  PROC DrawPart24()
    MoveL Offs(pOrigin,272.74,80.44,0.00),v40,z0,tPen\WObj:=wPaper;
    MoveL Offs(pOrigin,271.25,97.44,0.00),v40,z0,tPen\WObj:=wPaper;
    MoveL Offs(pOrigin,271.04,102.96,0.00),v40,z0,tPen\WObj:=wPaper;
    MoveL Offs(pOrigin,271.25,114.65,0.00),v40,z0,tPen\WObj:=wPaper;
    MoveL Offs(pOrigin,272.95,133.56,0.00),v40,z0,tPen\WObj:=wPaper;
    MoveL Offs(pOrigin,275.92,151.84,0.00),v40,z0,tPen\WObj:=wPaper;
    MoveL Offs(pOrigin,275.71,152.69,0.00),v40,z0,tPen\WObj:=wPaper;
    MoveL Offs(pOrigin,275.71,152.69,0.00),v40,z0,tPen\WObj:=wPaper;
    MoveL Offs(pOrigin,276.35,154.39,0.00),v40,z0,tPen\WObj:=wPaper;
    MoveL Offs(pOrigin,280.39,173.73,0.00),v40,z0,tPen\WObj:=wPaper;
    MoveL Offs(pOrigin,280.39,175.43,0.00),v40,z0,tPen\WObj:=wPaper;
    MoveL Offs(pOrigin,281.24,177.12,0.00),v40,z0,tPen\WObj:=wPaper;
    MoveL Offs(pOrigin,286.76,199.01,0.00),v40,z0,tPen\WObj:=wPaper;
    MoveL Offs(pOrigin,286.76,199.01,0.00),v40,z0,tPen\WObj:=wPaper;
    MoveL Offs(pOrigin,288.25,206.66,0.00),v40,z0,tPen\WObj:=wPaper;
    MoveL Offs(pOrigin,289.10,213.46,0.00),v40,z0,tPen\WObj:=wPaper;
    MoveL Offs(pOrigin,289.10,221.32,0.00),v40,z0,tPen\WObj:=wPaper;
    MoveL Offs(pOrigin,288.82,222.39,0.00),v40,z0,tPen\WObj:=wPaper;
    MoveL Offs(pOrigin,288.25,222.81,0.00),v40,fine,tPen\WObj:=wPaper;
    MoveL Offs(pOrigin,288.25,222.81,6.00),v60,z5,tPen\WObj:=wPaper;
    MoveL Offs(pOrigin,287.19,224.30,6.00),vTravel,z5,tPen\WObj:=wPaper;
    MoveL Offs(pOrigin,287.19,224.30,0.00),v60,z0,tPen\WObj:=wPaper;
    MoveL Offs(pOrigin,287.61,224.51,0.00),v40,z0,tPen\WObj:=wPaper;
    MoveL Offs(pOrigin,287.19,224.30,0.00),v40,fine,tPen\WObj:=wPaper;
    MoveL Offs(pOrigin,287.19,224.30,6.00),v60,z5,tPen\WObj:=wPaper;
    MoveL Offs(pOrigin,296.11,217.29,6.00),vTravel,z5,tPen\WObj:=wPaper;
    MoveL Offs(pOrigin,296.11,217.29,0.00),v60,z0,tPen\WObj:=wPaper;
    MoveL Offs(pOrigin,294.41,218.99,0.00),v40,z0,tPen\WObj:=wPaper;
    MoveL Offs(pOrigin,296.11,217.29,0.00),v40,fine,tPen\WObj:=wPaper;
    MoveL Offs(pOrigin,296.11,217.29,6.00),v60,z5,tPen\WObj:=wPaper;
    MoveL Offs(pOrigin,297.81,215.59,6.00),vTravel,z5,tPen\WObj:=wPaper;
    MoveL Offs(pOrigin,297.81,215.59,0.00),v60,z0,tPen\WObj:=wPaper;
    MoveL Offs(pOrigin,296.33,217.07,0.00),v40,z0,tPen\WObj:=wPaper;
    MoveL Offs(pOrigin,297.81,215.59,0.00),v40,fine,tPen\WObj:=wPaper;
    MoveL Offs(pOrigin,297.81,215.59,6.00),v60,z5,tPen\WObj:=wPaper;
    MoveL Offs(pOrigin,299.73,213.68,6.00),vTravel,z5,tPen\WObj:=wPaper;
    MoveL Offs(pOrigin,299.73,213.68,0.00),v60,z0,tPen\WObj:=wPaper;
    MoveL Offs(pOrigin,298.02,215.38,0.00),v40,z0,tPen\WObj:=wPaper;
    MoveL Offs(pOrigin,299.73,213.68,0.00),v40,fine,tPen\WObj:=wPaper;
    MoveL Offs(pOrigin,299.73,213.68,6.00),v60,z5,tPen\WObj:=wPaper;
    MoveL Offs(pOrigin,302.06,212.40,6.00),vTravel,z5,tPen\WObj:=wPaper;
    MoveL Offs(pOrigin,302.06,212.40,0.00),v60,z0,tPen\WObj:=wPaper;
    MoveL Offs(pOrigin,300.36,213.25,0.00),v40,z0,tPen\WObj:=wPaper;
    MoveL Offs(pOrigin,293.77,219.84,0.00),v40,z0,tPen\WObj:=wPaper;
    MoveL Offs(pOrigin,290.59,223.88,0.00),v40,z0,tPen\WObj:=wPaper;
    MoveL Offs(pOrigin,288.32,225.36,0.00),v40,z0,tPen\WObj:=wPaper;
    MoveL Offs(pOrigin,288.46,226.64,0.00),v40,z0,tPen\WObj:=wPaper;
    MoveL Offs(pOrigin,290.80,233.65,0.00),v40,z0,tPen\WObj:=wPaper;
    MoveL Offs(pOrigin,291.44,238.54,0.00),v40,fine,tPen\WObj:=wPaper;
    MoveL Offs(pOrigin,291.44,238.54,6.00),v60,z5,tPen\WObj:=wPaper;
    MoveL Offs(pOrigin,296.11,238.96,6.00),vTravel,z5,tPen\WObj:=wPaper;
    MoveL Offs(pOrigin,296.11,238.96,0.00),v60,z0,tPen\WObj:=wPaper;
    MoveL Offs(pOrigin,296.54,239.39,0.00),v40,z0,tPen\WObj:=wPaper;
    MoveL Offs(pOrigin,296.11,238.96,0.00),v40,fine,tPen\WObj:=wPaper;
    MoveL Offs(pOrigin,296.11,238.96,6.00),v60,z5,tPen\WObj:=wPaper;
    MoveL Offs(pOrigin,298.24,258.51,6.00),vTravel,z5,tPen\WObj:=wPaper;
    MoveL Offs(pOrigin,298.24,258.51,0.00),v60,z0,tPen\WObj:=wPaper;
    MoveL Offs(pOrigin,296.54,265.52,0.00),v40,fine,tPen\WObj:=wPaper;
    MoveL Offs(pOrigin,296.54,265.52,6.00),v60,z5,tPen\WObj:=wPaper;
    MoveL Offs(pOrigin,293.77,269.77,6.00),vTravel,z5,tPen\WObj:=wPaper;
    MoveL Offs(pOrigin,293.77,269.77,0.00),v60,z0,tPen\WObj:=wPaper;
    MoveL Offs(pOrigin,294.20,270.20,0.00),v40,z0,tPen\WObj:=wPaper;
    MoveL Offs(pOrigin,293.77,269.77,0.00),v40,fine,tPen\WObj:=wPaper;
    MoveL Offs(pOrigin,293.77,269.77,6.00),v60,z5,tPen\WObj:=wPaper;
    MoveL Offs(pOrigin,289.10,272.33,6.00),vTravel,z5,tPen\WObj:=wPaper;
    MoveL Offs(pOrigin,289.10,272.33,0.00),v60,z0,tPen\WObj:=wPaper;
    MoveL Offs(pOrigin,288.25,272.96,0.00),v40,z0,tPen\WObj:=wPaper;
    MoveL Offs(pOrigin,283.36,274.02,0.00),v40,z0,tPen\WObj:=wPaper;
    MoveL Offs(pOrigin,282.30,276.15,0.00),v40,z0,tPen\WObj:=wPaper;
    MoveL Offs(pOrigin,282.30,277.64,0.00),v40,z0,tPen\WObj:=wPaper;
    MoveL Offs(pOrigin,282.30,277.64,0.00),v40,z0,tPen\WObj:=wPaper;
    MoveL Offs(pOrigin,281.45,278.70,0.00),v40,z0,tPen\WObj:=wPaper;
    MoveL Offs(pOrigin,281.45,279.76,0.00),v40,z0,tPen\WObj:=wPaper;
    MoveL Offs(pOrigin,281.45,279.76,0.00),v40,z0,tPen\WObj:=wPaper;
    MoveL Offs(pOrigin,281.88,280.61,0.00),v40,z0,tPen\WObj:=wPaper;
    MoveL Offs(pOrigin,281.88,281.46,0.00),v40,z0,tPen\WObj:=wPaper;
    MoveL Offs(pOrigin,281.52,282.95,0.00),v40,z0,tPen\WObj:=wPaper;
    MoveL Offs(pOrigin,279.33,286.56,0.00),v40,fine,tPen\WObj:=wPaper;
    MoveL Offs(pOrigin,279.33,286.56,6.00),v60,z5,tPen\WObj:=wPaper;
    MoveL Offs(pOrigin,278.90,284.86,6.00),vTravel,z5,tPen\WObj:=wPaper;
    MoveL Offs(pOrigin,278.90,284.86,0.00),v60,z0,tPen\WObj:=wPaper;
    MoveL Offs(pOrigin,280.81,281.89,0.00),v40,z0,tPen\WObj:=wPaper;
    MoveL Offs(pOrigin,281.88,281.46,0.00),v40,z0,tPen\WObj:=wPaper;
    MoveL Offs(pOrigin,281.88,281.46,0.00),v40,z0,tPen\WObj:=wPaper;
    MoveL Offs(pOrigin,281.95,280.83,0.00),v40,z0,tPen\WObj:=wPaper;
    MoveL Offs(pOrigin,282.87,280.33,0.00),v40,z0,tPen\WObj:=wPaper;
    MoveL Offs(pOrigin,284.64,278.27,0.00),v40,z0,tPen\WObj:=wPaper;
    MoveL Offs(pOrigin,285.49,276.58,0.00),v40,z0,tPen\WObj:=wPaper;
    MoveL Offs(pOrigin,285.49,276.58,0.00),v40,z0,tPen\WObj:=wPaper;
    MoveL Offs(pOrigin,286.34,275.87,0.00),v40,z0,tPen\WObj:=wPaper;
    MoveL Offs(pOrigin,288.89,275.30,0.00),v40,z0,tPen\WObj:=wPaper;
    MoveL Offs(pOrigin,288.89,275.30,0.00),v40,z0,tPen\WObj:=wPaper;
    MoveL Offs(pOrigin,289.31,275.73,0.00),v40,z0,tPen\WObj:=wPaper;
    MoveL Offs(pOrigin,290.38,275.73,0.00),v40,z0,tPen\WObj:=wPaper;
    MoveL Offs(pOrigin,290.80,276.15,0.00),v40,fine,tPen\WObj:=wPaper;
    MoveL Offs(pOrigin,290.80,276.15,6.00),v60,z5,tPen\WObj:=wPaper;
    MoveL Offs(pOrigin,292.71,275.94,6.00),vTravel,z5,tPen\WObj:=wPaper;
    MoveL Offs(pOrigin,292.71,275.94,0.00),v60,z0,tPen\WObj:=wPaper;
    MoveL Offs(pOrigin,291.65,274.80,0.00),v40,z0,tPen\WObj:=wPaper;
    MoveL Offs(pOrigin,290.16,274.45,0.00),v40,z0,tPen\WObj:=wPaper;
    MoveL Offs(pOrigin,289.52,274.52,0.00),v40,z0,tPen\WObj:=wPaper;
    MoveL Offs(pOrigin,288.89,275.30,0.00),v40,fine,tPen\WObj:=wPaper;
    MoveL Offs(pOrigin,288.89,275.30,6.00),v60,z5,tPen\WObj:=wPaper;
    MoveL Offs(pOrigin,289.31,277.42,6.00),vTravel,z5,tPen\WObj:=wPaper;
    MoveL Offs(pOrigin,289.31,277.42,0.00),v60,z0,tPen\WObj:=wPaper;
    MoveL Offs(pOrigin,288.04,277.57,0.00),v40,z0,tPen\WObj:=wPaper;
    MoveL Offs(pOrigin,286.55,278.70,0.00),v40,z0,tPen\WObj:=wPaper;
    MoveL Offs(pOrigin,286.34,280.61,0.00),v40,z0,tPen\WObj:=wPaper;
    MoveL Offs(pOrigin,286.34,280.61,0.00),v40,z0,tPen\WObj:=wPaper;
    MoveL Offs(pOrigin,284.64,281.89,0.00),v40,z0,tPen\WObj:=wPaper;
    MoveL Offs(pOrigin,283.36,283.38,0.00),v40,z0,tPen\WObj:=wPaper;
    MoveL Offs(pOrigin,282.94,285.08,0.00),v40,z0,tPen\WObj:=wPaper;
    MoveL Offs(pOrigin,282.94,285.08,0.00),v40,z0,tPen\WObj:=wPaper;
    MoveL Offs(pOrigin,281.31,288.05,0.00),v40,z0,tPen\WObj:=wPaper;
    MoveL Offs(pOrigin,282.51,289.11,0.00),v40,z0,tPen\WObj:=wPaper;
    MoveL Offs(pOrigin,282.51,289.11,0.00),v40,z0,tPen\WObj:=wPaper;
    MoveL Offs(pOrigin,282.51,289.75,0.00),v40,z0,tPen\WObj:=wPaper;
    MoveL Offs(pOrigin,281.88,290.39,0.00),v40,z0,tPen\WObj:=wPaper;
    MoveL Offs(pOrigin,282.09,290.17,0.00),v40,z0,tPen\WObj:=wPaper;
    MoveL Offs(pOrigin,281.66,290.81,0.00),v40,z0,tPen\WObj:=wPaper;
  ENDPROC

  PROC DrawPart25()
    MoveL Offs(pOrigin,280.81,294.00,0.00),v40,z0,tPen\WObj:=wPaper;
    MoveL Offs(pOrigin,280.81,294.00,0.00),v40,z0,tPen\WObj:=wPaper;
    MoveL Offs(pOrigin,279.54,294.85,0.00),v40,z0,tPen\WObj:=wPaper;
    MoveL Offs(pOrigin,279.11,295.06,0.00),v40,z0,tPen\WObj:=wPaper;
    MoveL Offs(pOrigin,279.33,294.85,0.00),v40,z0,tPen\WObj:=wPaper;
    MoveL Offs(pOrigin,279.54,295.06,0.00),v40,z0,tPen\WObj:=wPaper;
    MoveL Offs(pOrigin,279.33,295.49,0.00),v40,z0,tPen\WObj:=wPaper;
    MoveL Offs(pOrigin,278.90,295.27,0.00),v40,z0,tPen\WObj:=wPaper;
    MoveL Offs(pOrigin,279.25,295.91,0.00),v40,z0,tPen\WObj:=wPaper;
    MoveL Offs(pOrigin,278.26,296.98,0.00),v40,z0,tPen\WObj:=wPaper;
    MoveL Offs(pOrigin,277.84,297.19,0.00),v40,z0,tPen\WObj:=wPaper;
    MoveL Offs(pOrigin,276.77,298.04,0.00),v40,fine,tPen\WObj:=wPaper;
    MoveL Offs(pOrigin,276.77,298.04,6.00),v60,z5,tPen\WObj:=wPaper;
    MoveL Offs(pOrigin,277.41,299.52,6.00),vTravel,z5,tPen\WObj:=wPaper;
    MoveL Offs(pOrigin,277.41,299.52,0.00),v60,z0,tPen\WObj:=wPaper;
    MoveL Offs(pOrigin,277.41,299.31,0.00),v40,z0,tPen\WObj:=wPaper;
    MoveL Offs(pOrigin,276.99,299.52,0.00),v40,z0,tPen\WObj:=wPaper;
    MoveL Offs(pOrigin,276.35,300.59,0.00),v40,z0,tPen\WObj:=wPaper;
    MoveL Offs(pOrigin,275.71,300.80,0.00),v40,fine,tPen\WObj:=wPaper;
    MoveL Offs(pOrigin,275.71,300.80,6.00),v60,z5,tPen\WObj:=wPaper;
    MoveL Offs(pOrigin,276.14,302.29,6.00),vTravel,z5,tPen\WObj:=wPaper;
    MoveL Offs(pOrigin,276.14,302.29,0.00),v60,z0,tPen\WObj:=wPaper;
    MoveL Offs(pOrigin,272.74,303.56,0.00),v40,fine,tPen\WObj:=wPaper;
    MoveL Offs(pOrigin,272.74,303.56,6.00),v60,z5,tPen\WObj:=wPaper;
    MoveL Offs(pOrigin,271.04,305.26,6.00),vTravel,z5,tPen\WObj:=wPaper;
    MoveL Offs(pOrigin,271.04,305.26,0.00),v60,z0,tPen\WObj:=wPaper;
    MoveL Offs(pOrigin,275.50,303.85,0.00),v40,z0,tPen\WObj:=wPaper;
    MoveL Offs(pOrigin,276.14,304.41,0.00),v40,z0,tPen\WObj:=wPaper;
    MoveL Offs(pOrigin,276.35,303.99,0.00),v40,z0,tPen\WObj:=wPaper;
    MoveL Offs(pOrigin,276.77,304.20,0.00),v40,z0,tPen\WObj:=wPaper;
    MoveL Offs(pOrigin,276.35,303.99,0.00),v40,z0,tPen\WObj:=wPaper;
    MoveL Offs(pOrigin,276.77,303.77,0.00),v40,z0,tPen\WObj:=wPaper;
    MoveL Offs(pOrigin,277.20,303.56,0.00),v40,z0,tPen\WObj:=wPaper;
    MoveL Offs(pOrigin,276.77,303.77,0.00),v40,z0,tPen\WObj:=wPaper;
    MoveL Offs(pOrigin,277.41,303.56,0.00),v40,z0,tPen\WObj:=wPaper;
    MoveL Offs(pOrigin,279.11,302.50,0.00),v40,z0,tPen\WObj:=wPaper;
    MoveL Offs(pOrigin,277.41,303.56,0.00),v40,fine,tPen\WObj:=wPaper;
    MoveL Offs(pOrigin,277.41,303.56,6.00),v60,z5,tPen\WObj:=wPaper;
    MoveL Offs(pOrigin,276.77,305.48,6.00),vTravel,z5,tPen\WObj:=wPaper;
    MoveL Offs(pOrigin,276.77,305.48,0.00),v60,z0,tPen\WObj:=wPaper;
    MoveL Offs(pOrigin,276.70,304.41,0.00),v40,z0,tPen\WObj:=wPaper;
    MoveL Offs(pOrigin,276.14,303.77,0.00),v40,z0,tPen\WObj:=wPaper;
    MoveL Offs(pOrigin,276.14,302.71,0.00),v40,z0,tPen\WObj:=wPaper;
    MoveL Offs(pOrigin,276.56,301.86,0.00),v40,z0,tPen\WObj:=wPaper;
    MoveL Offs(pOrigin,278.12,300.38,0.00),v40,z0,tPen\WObj:=wPaper;
    MoveL Offs(pOrigin,278.19,299.95,0.00),v40,z0,tPen\WObj:=wPaper;
    MoveL Offs(pOrigin,277.84,299.74,0.00),v40,fine,tPen\WObj:=wPaper;
    MoveL Offs(pOrigin,277.84,299.74,6.00),v60,z5,tPen\WObj:=wPaper;
    MoveL Offs(pOrigin,279.33,299.52,6.00),vTravel,z5,tPen\WObj:=wPaper;
    MoveL Offs(pOrigin,279.33,299.52,0.00),v60,z0,tPen\WObj:=wPaper;
    MoveL Offs(pOrigin,278.90,298.89,0.00),v40,z0,tPen\WObj:=wPaper;
    MoveL Offs(pOrigin,279.96,297.40,0.00),v40,z0,tPen\WObj:=wPaper;
    MoveL Offs(pOrigin,281.45,295.98,0.00),v40,z0,tPen\WObj:=wPaper;
    MoveL Offs(pOrigin,282.30,295.63,0.00),v40,z0,tPen\WObj:=wPaper;
    MoveL Offs(pOrigin,284.64,293.15,0.00),v40,z0,tPen\WObj:=wPaper;
    MoveL Offs(pOrigin,289.95,290.39,0.00),v40,fine,tPen\WObj:=wPaper;
    MoveL Offs(pOrigin,289.95,290.39,6.00),v60,z5,tPen\WObj:=wPaper;
    MoveL Offs(pOrigin,286.55,290.17,6.00),vTravel,z5,tPen\WObj:=wPaper;
    MoveL Offs(pOrigin,286.55,290.17,0.00),v60,z0,tPen\WObj:=wPaper;
    MoveL Offs(pOrigin,284.64,291.24,0.00),v40,z0,tPen\WObj:=wPaper;
    MoveL Offs(pOrigin,284.21,291.45,0.00),v40,z0,tPen\WObj:=wPaper;
    MoveL Offs(pOrigin,282.30,293.50,0.00),v40,z0,tPen\WObj:=wPaper;
    MoveL Offs(pOrigin,281.02,294.00,0.00),v40,z0,tPen\WObj:=wPaper;
    MoveL Offs(pOrigin,280.81,294.00,0.00),v40,z0,tPen\WObj:=wPaper;
    MoveL Offs(pOrigin,281.24,294.64,0.00),v40,z0,tPen\WObj:=wPaper;
    MoveL Offs(pOrigin,281.24,295.91,0.00),v40,fine,tPen\WObj:=wPaper;
    MoveL Offs(pOrigin,281.24,295.91,6.00),v60,z5,tPen\WObj:=wPaper;
    MoveL Offs(pOrigin,283.36,294.21,6.00),vTravel,z5,tPen\WObj:=wPaper;
    MoveL Offs(pOrigin,283.36,294.21,0.00),v60,z0,tPen\WObj:=wPaper;
    MoveL Offs(pOrigin,282.73,294.85,0.00),v40,z0,tPen\WObj:=wPaper;
    MoveL Offs(pOrigin,283.36,294.21,0.00),v40,fine,tPen\WObj:=wPaper;
    MoveL Offs(pOrigin,283.36,294.21,6.00),v60,z5,tPen\WObj:=wPaper;
    MoveL Offs(pOrigin,284.00,296.12,6.00),vTravel,z5,tPen\WObj:=wPaper;
    MoveL Offs(pOrigin,284.00,296.12,0.00),v60,z0,tPen\WObj:=wPaper;
    MoveL Offs(pOrigin,282.51,297.61,0.00),v40,z0,tPen\WObj:=wPaper;
    MoveL Offs(pOrigin,284.00,296.12,0.00),v40,fine,tPen\WObj:=wPaper;
    MoveL Offs(pOrigin,284.00,296.12,6.00),v60,z5,tPen\WObj:=wPaper;
    MoveL Offs(pOrigin,285.70,294.64,6.00),vTravel,z5,tPen\WObj:=wPaper;
    MoveL Offs(pOrigin,285.70,294.64,0.00),v60,z0,tPen\WObj:=wPaper;
    MoveL Offs(pOrigin,284.64,295.70,0.00),v40,z0,tPen\WObj:=wPaper;
    MoveL Offs(pOrigin,285.70,294.64,0.00),v40,fine,tPen\WObj:=wPaper;
    MoveL Offs(pOrigin,285.70,294.64,6.00),v60,z5,tPen\WObj:=wPaper;
    MoveL Offs(pOrigin,287.61,294.21,6.00),vTravel,z5,tPen\WObj:=wPaper;
    MoveL Offs(pOrigin,287.61,294.21,0.00),v60,z0,tPen\WObj:=wPaper;
    MoveL Offs(pOrigin,287.83,295.42,0.00),v40,z0,tPen\WObj:=wPaper;
    MoveL Offs(pOrigin,291.01,295.06,0.00),v40,z0,tPen\WObj:=wPaper;
    MoveL Offs(pOrigin,292.08,295.42,0.00),v40,z0,tPen\WObj:=wPaper;
    MoveL Offs(pOrigin,292.50,295.91,0.00),v40,z0,tPen\WObj:=wPaper;
    MoveL Offs(pOrigin,292.50,295.91,0.00),v40,z0,tPen\WObj:=wPaper;
    MoveL Offs(pOrigin,296.54,297.40,0.00),v40,z0,tPen\WObj:=wPaper;
    MoveL Offs(pOrigin,296.54,297.40,0.00),v40,z0,tPen\WObj:=wPaper;
    MoveL Offs(pOrigin,296.54,299.31,0.00),v40,z0,tPen\WObj:=wPaper;
    MoveL Offs(pOrigin,296.11,299.74,0.00),v40,z0,tPen\WObj:=wPaper;
    MoveL Offs(pOrigin,296.11,299.74,0.00),v40,z0,tPen\WObj:=wPaper;
    MoveL Offs(pOrigin,296.11,300.80,0.00),v40,z0,tPen\WObj:=wPaper;
    MoveL Offs(pOrigin,296.11,300.80,0.00),v40,z0,tPen\WObj:=wPaper;
    MoveL Offs(pOrigin,295.69,303.14,0.00),v40,z0,tPen\WObj:=wPaper;
    MoveL Offs(pOrigin,295.69,303.14,0.00),v40,z0,tPen\WObj:=wPaper;
    MoveL Offs(pOrigin,295.90,303.77,0.00),v40,z0,tPen\WObj:=wPaper;
    MoveL Offs(pOrigin,295.12,305.69,0.00),v40,z0,tPen\WObj:=wPaper;
    MoveL Offs(pOrigin,293.56,306.54,0.00),v40,z0,tPen\WObj:=wPaper;
    MoveL Offs(pOrigin,293.07,308.45,0.00),v40,z0,tPen\WObj:=wPaper;
    MoveL Offs(pOrigin,292.15,309.30,0.00),v40,z0,tPen\WObj:=wPaper;
    MoveL Offs(pOrigin,291.93,310.36,0.00),v40,z0,tPen\WObj:=wPaper;
    MoveL Offs(pOrigin,292.29,311.00,0.00),v40,z0,tPen\WObj:=wPaper;
    MoveL Offs(pOrigin,292.29,312.06,0.00),v40,z0,tPen\WObj:=wPaper;
    MoveL Offs(pOrigin,291.86,313.12,0.00),v40,z0,tPen\WObj:=wPaper;
    MoveL Offs(pOrigin,291.86,313.12,0.00),v40,z0,tPen\WObj:=wPaper;
    MoveL Offs(pOrigin,290.80,312.91,0.00),v40,z0,tPen\WObj:=wPaper;
    MoveL Offs(pOrigin,290.80,312.91,0.00),v40,z0,tPen\WObj:=wPaper;
    MoveL Offs(pOrigin,290.80,313.34,0.00),v40,z0,tPen\WObj:=wPaper;
    MoveL Offs(pOrigin,291.44,313.55,0.00),v40,z0,tPen\WObj:=wPaper;
    MoveL Offs(pOrigin,291.44,313.55,0.00),v40,z0,tPen\WObj:=wPaper;
    MoveL Offs(pOrigin,291.44,314.19,0.00),v40,z0,tPen\WObj:=wPaper;
    MoveL Offs(pOrigin,290.59,314.40,0.00),v40,fine,tPen\WObj:=wPaper;
    MoveL Offs(pOrigin,290.59,314.40,6.00),v60,z5,tPen\WObj:=wPaper;
    MoveL Offs(pOrigin,290.80,312.91,6.00),vTravel,z5,tPen\WObj:=wPaper;
    MoveL Offs(pOrigin,290.80,312.91,0.00),v60,z0,tPen\WObj:=wPaper;
    MoveL Offs(pOrigin,290.59,312.06,0.00),v40,z0,tPen\WObj:=wPaper;
    MoveL Offs(pOrigin,290.87,311.21,0.00),v40,z0,tPen\WObj:=wPaper;
  ENDPROC

  PROC DrawPart26()
    MoveL Offs(pOrigin,291.86,310.58,0.00),v40,fine,tPen\WObj:=wPaper;
    MoveL Offs(pOrigin,291.86,310.58,6.00),v60,z5,tPen\WObj:=wPaper;
    MoveL Offs(pOrigin,292.08,309.09,6.00),vTravel,z5,tPen\WObj:=wPaper;
    MoveL Offs(pOrigin,292.08,309.09,0.00),v60,z0,tPen\WObj:=wPaper;
    MoveL Offs(pOrigin,291.51,308.45,0.00),v40,z0,tPen\WObj:=wPaper;
    MoveL Offs(pOrigin,291.01,306.54,0.00),v40,z0,tPen\WObj:=wPaper;
    MoveL Offs(pOrigin,291.01,306.54,0.00),v40,z0,tPen\WObj:=wPaper;
    MoveL Offs(pOrigin,289.88,307.39,0.00),v40,z0,tPen\WObj:=wPaper;
    MoveL Offs(pOrigin,288.75,310.15,0.00),v40,z0,tPen\WObj:=wPaper;
    MoveL Offs(pOrigin,287.12,312.49,0.00),v40,z0,tPen\WObj:=wPaper;
    MoveL Offs(pOrigin,285.49,313.62,0.00),v40,z0,tPen\WObj:=wPaper;
    MoveL Offs(pOrigin,283.79,314.19,0.00),v40,z0,tPen\WObj:=wPaper;
    MoveL Offs(pOrigin,280.17,313.69,0.00),v40,z0,tPen\WObj:=wPaper;
    MoveL Offs(pOrigin,276.99,312.13,0.00),v40,z0,tPen\WObj:=wPaper;
    MoveL Offs(pOrigin,275.50,311.00,0.00),v40,z0,tPen\WObj:=wPaper;
    MoveL Offs(pOrigin,271.46,311.00,0.00),v40,z0,tPen\WObj:=wPaper;
    MoveL Offs(pOrigin,270.61,311.64,0.00),v40,z0,tPen\WObj:=wPaper;
    MoveL Offs(pOrigin,270.61,311.64,0.00),v40,z0,tPen\WObj:=wPaper;
    MoveL Offs(pOrigin,271.04,312.91,0.00),v40,z0,tPen\WObj:=wPaper;
    MoveL Offs(pOrigin,271.04,312.91,0.00),v40,z0,tPen\WObj:=wPaper;
    MoveL Offs(pOrigin,276.77,314.40,0.00),v40,z0,tPen\WObj:=wPaper;
    MoveL Offs(pOrigin,276.77,314.40,0.00),v40,z0,tPen\WObj:=wPaper;
    MoveL Offs(pOrigin,278.26,314.19,0.00),v40,z0,tPen\WObj:=wPaper;
    MoveL Offs(pOrigin,278.90,314.40,0.00),v40,fine,tPen\WObj:=wPaper;
    MoveL Offs(pOrigin,278.90,314.40,6.00),v60,z5,tPen\WObj:=wPaper;
    MoveL Offs(pOrigin,276.77,314.40,6.00),vTravel,z5,tPen\WObj:=wPaper;
    MoveL Offs(pOrigin,276.77,314.40,0.00),v60,z0,tPen\WObj:=wPaper;
    MoveL Offs(pOrigin,278.26,315.60,0.00),v40,z0,tPen\WObj:=wPaper;
    MoveL Offs(pOrigin,281.24,316.74,0.00),v40,z0,tPen\WObj:=wPaper;
    MoveL Offs(pOrigin,284.64,316.95,0.00),v40,z0,tPen\WObj:=wPaper;
    MoveL Offs(pOrigin,286.34,316.38,0.00),v40,z0,tPen\WObj:=wPaper;
    MoveL Offs(pOrigin,289.95,313.48,0.00),v40,z0,tPen\WObj:=wPaper;
    MoveL Offs(pOrigin,290.30,313.76,0.00),v40,z0,tPen\WObj:=wPaper;
    MoveL Offs(pOrigin,290.52,314.83,0.00),v40,z0,tPen\WObj:=wPaper;
    MoveL Offs(pOrigin,288.89,317.80,0.00),v40,z0,tPen\WObj:=wPaper;
    MoveL Offs(pOrigin,288.89,317.80,0.00),v40,z0,tPen\WObj:=wPaper;
    MoveL Offs(pOrigin,288.53,319.92,0.00),v40,z0,tPen\WObj:=wPaper;
    MoveL Offs(pOrigin,286.98,322.05,0.00),v40,z0,tPen\WObj:=wPaper;
    MoveL Offs(pOrigin,284.42,324.60,0.00),v40,z0,tPen\WObj:=wPaper;
    MoveL Offs(pOrigin,280.81,326.58,0.00),v40,z0,tPen\WObj:=wPaper;
    MoveL Offs(pOrigin,275.08,327.86,0.00),v40,z0,tPen\WObj:=wPaper;
    MoveL Offs(pOrigin,272.10,331.54,0.00),v40,z0,tPen\WObj:=wPaper;
    MoveL Offs(pOrigin,268.70,334.02,0.00),v40,z0,tPen\WObj:=wPaper;
    MoveL Offs(pOrigin,267.42,334.38,0.00),v40,z0,tPen\WObj:=wPaper;
    MoveL Offs(pOrigin,267.42,334.38,0.00),v40,z0,tPen\WObj:=wPaper;
    MoveL Offs(pOrigin,267.21,333.10,0.00),v40,z0,tPen\WObj:=wPaper;
    MoveL Offs(pOrigin,267.21,333.10,0.00),v40,z0,tPen\WObj:=wPaper;
    MoveL Offs(pOrigin,265.30,333.74,0.00),v40,z0,tPen\WObj:=wPaper;
    MoveL Offs(pOrigin,265.30,333.52,0.00),v40,z0,tPen\WObj:=wPaper;
    MoveL Offs(pOrigin,265.30,333.52,0.00),v40,z0,tPen\WObj:=wPaper;
    MoveL Offs(pOrigin,266.72,329.27,0.00),v40,z0,tPen\WObj:=wPaper;
    MoveL Offs(pOrigin,267.42,328.64,0.00),v40,z0,tPen\WObj:=wPaper;
    MoveL Offs(pOrigin,267.42,328.64,0.00),v40,z0,tPen\WObj:=wPaper;
    MoveL Offs(pOrigin,265.80,325.02,0.00),v40,z0,tPen\WObj:=wPaper;
    MoveL Offs(pOrigin,263.88,322.69,0.00),v40,z0,tPen\WObj:=wPaper;
    MoveL Offs(pOrigin,263.81,322.05,0.00),v40,z0,tPen\WObj:=wPaper;
    MoveL Offs(pOrigin,263.81,322.05,0.00),v40,z0,tPen\WObj:=wPaper;
    MoveL Offs(pOrigin,264.02,321.84,0.00),v40,z0,tPen\WObj:=wPaper;
    MoveL Offs(pOrigin,264.88,322.05,0.00),v40,z0,tPen\WObj:=wPaper;
    MoveL Offs(pOrigin,265.30,321.62,0.00),v40,z0,tPen\WObj:=wPaper;
    MoveL Offs(pOrigin,265.30,321.62,0.00),v40,z0,tPen\WObj:=wPaper;
    MoveL Offs(pOrigin,267.21,323.54,0.00),v40,z0,tPen\WObj:=wPaper;
    MoveL Offs(pOrigin,268.27,325.24,0.00),v40,z0,tPen\WObj:=wPaper;
    MoveL Offs(pOrigin,269.12,325.66,0.00),v40,z0,tPen\WObj:=wPaper;
    MoveL Offs(pOrigin,269.55,326.30,0.00),v40,fine,tPen\WObj:=wPaper;
    MoveL Offs(pOrigin,269.55,326.30,6.00),v60,z5,tPen\WObj:=wPaper;
    MoveL Offs(pOrigin,268.06,325.24,6.00),vTravel,z5,tPen\WObj:=wPaper;
    MoveL Offs(pOrigin,268.06,325.24,0.00),v60,z0,tPen\WObj:=wPaper;
    MoveL Offs(pOrigin,268.06,326.94,0.00),v40,z0,tPen\WObj:=wPaper;
    MoveL Offs(pOrigin,267.42,327.79,0.00),v40,z0,tPen\WObj:=wPaper;
    MoveL Offs(pOrigin,267.42,328.64,0.00),v40,z0,tPen\WObj:=wPaper;
    MoveL Offs(pOrigin,267.99,329.06,0.00),v40,z0,tPen\WObj:=wPaper;
    MoveL Offs(pOrigin,268.27,331.19,0.00),v40,z0,tPen\WObj:=wPaper;
    MoveL Offs(pOrigin,268.27,331.19,0.00),v40,z0,tPen\WObj:=wPaper;
    MoveL Offs(pOrigin,269.34,330.98,0.00),v40,z0,tPen\WObj:=wPaper;
    MoveL Offs(pOrigin,269.34,330.98,0.00),v40,z0,tPen\WObj:=wPaper;
    MoveL Offs(pOrigin,270.19,330.83,0.00),v40,z0,tPen\WObj:=wPaper;
    MoveL Offs(pOrigin,271.25,329.91,0.00),v40,z0,tPen\WObj:=wPaper;
    MoveL Offs(pOrigin,271.89,328.21,0.00),v40,z0,tPen\WObj:=wPaper;
    MoveL Offs(pOrigin,271.89,328.21,0.00),v40,z0,tPen\WObj:=wPaper;
    MoveL Offs(pOrigin,271.46,326.80,0.00),v40,z0,tPen\WObj:=wPaper;
    MoveL Offs(pOrigin,269.62,326.51,0.00),v40,z0,tPen\WObj:=wPaper;
    MoveL Offs(pOrigin,269.76,329.27,0.00),v40,z0,tPen\WObj:=wPaper;
    MoveL Offs(pOrigin,269.34,330.98,0.00),v40,z0,tPen\WObj:=wPaper;
    MoveL Offs(pOrigin,268.27,331.19,0.00),v40,z0,tPen\WObj:=wPaper;
    MoveL Offs(pOrigin,267.21,333.10,0.00),v40,fine,tPen\WObj:=wPaper;
    MoveL Offs(pOrigin,267.21,333.10,6.00),v60,z5,tPen\WObj:=wPaper;
    MoveL Offs(pOrigin,267.42,334.38,6.00),vTravel,z5,tPen\WObj:=wPaper;
    MoveL Offs(pOrigin,267.42,334.38,0.00),v60,z0,tPen\WObj:=wPaper;
    MoveL Offs(pOrigin,265.94,335.23,0.00),v40,z0,tPen\WObj:=wPaper;
    MoveL Offs(pOrigin,265.73,335.65,0.00),v40,z0,tPen\WObj:=wPaper;
    MoveL Offs(pOrigin,265.94,335.44,0.00),v40,z0,tPen\WObj:=wPaper;
    MoveL Offs(pOrigin,265.51,335.65,0.00),v40,z0,tPen\WObj:=wPaper;
    MoveL Offs(pOrigin,263.81,336.29,0.00),v40,z0,tPen\WObj:=wPaper;
    MoveL Offs(pOrigin,262.96,336.08,0.00),v40,z0,tPen\WObj:=wPaper;
    MoveL Offs(pOrigin,262.96,336.08,0.00),v40,z0,tPen\WObj:=wPaper;
    MoveL Offs(pOrigin,263.60,334.80,0.00),v40,z0,tPen\WObj:=wPaper;
    MoveL Offs(pOrigin,265.30,333.52,0.00),v40,fine,tPen\WObj:=wPaper;
    MoveL Offs(pOrigin,265.30,333.52,6.00),v60,z5,tPen\WObj:=wPaper;
    MoveL Offs(pOrigin,262.96,336.08,6.00),vTravel,z5,tPen\WObj:=wPaper;
    MoveL Offs(pOrigin,262.96,336.08,0.00),v60,z0,tPen\WObj:=wPaper;
    MoveL Offs(pOrigin,260.41,336.92,0.00),v40,z0,tPen\WObj:=wPaper;
    MoveL Offs(pOrigin,259.14,336.92,0.00),v40,z0,tPen\WObj:=wPaper;
    MoveL Offs(pOrigin,259.14,336.92,0.00),v40,z0,tPen\WObj:=wPaper;
    MoveL Offs(pOrigin,259.42,336.08,0.00),v40,z0,tPen\WObj:=wPaper;
    MoveL Offs(pOrigin,262.11,333.52,0.00),v40,z0,tPen\WObj:=wPaper;
    MoveL Offs(pOrigin,263.60,330.34,0.00),v40,z0,tPen\WObj:=wPaper;
    MoveL Offs(pOrigin,263.60,327.58,0.00),v40,z0,tPen\WObj:=wPaper;
    MoveL Offs(pOrigin,262.89,325.24,0.00),v40,z0,tPen\WObj:=wPaper;
    MoveL Offs(pOrigin,261.69,323.33,0.00),v40,z0,tPen\WObj:=wPaper;
    MoveL Offs(pOrigin,260.20,321.84,0.00),v40,z0,tPen\WObj:=wPaper;
    MoveL Offs(pOrigin,259.56,320.56,0.00),v40,z0,tPen\WObj:=wPaper;
    MoveL Offs(pOrigin,259.56,320.56,0.00),v40,z0,tPen\WObj:=wPaper;
    MoveL Offs(pOrigin,260.41,320.35,0.00),v40,z0,tPen\WObj:=wPaper;
    MoveL Offs(pOrigin,261.48,320.70,0.00),v40,z0,tPen\WObj:=wPaper;
    MoveL Offs(pOrigin,263.81,322.05,0.00),v40,fine,tPen\WObj:=wPaper;
    MoveL Offs(pOrigin,263.81,322.05,6.00),v60,z5,tPen\WObj:=wPaper;
    MoveL Offs(pOrigin,265.30,321.62,6.00),vTravel,z5,tPen\WObj:=wPaper;
    MoveL Offs(pOrigin,265.30,321.62,0.00),v60,z0,tPen\WObj:=wPaper;
    MoveL Offs(pOrigin,263.39,319.08,0.00),v40,z0,tPen\WObj:=wPaper;
  ENDPROC

  PROC DrawPart27()
    MoveL Offs(pOrigin,263.39,319.08,0.00),v40,z0,tPen\WObj:=wPaper;
    MoveL Offs(pOrigin,259.77,317.66,0.00),v40,z0,tPen\WObj:=wPaper;
    MoveL Offs(pOrigin,259.35,316.95,0.00),v40,z0,tPen\WObj:=wPaper;
    MoveL Offs(pOrigin,259.35,316.95,0.00),v40,z0,tPen\WObj:=wPaper;
    MoveL Offs(pOrigin,259.99,316.52,0.00),v40,z0,tPen\WObj:=wPaper;
    MoveL Offs(pOrigin,262.96,316.95,0.00),v40,z0,tPen\WObj:=wPaper;
    MoveL Offs(pOrigin,264.02,316.10,0.00),v40,z0,tPen\WObj:=wPaper;
    MoveL Offs(pOrigin,264.02,316.10,0.00),v40,z0,tPen\WObj:=wPaper;
    MoveL Offs(pOrigin,266.15,316.52,0.00),v40,z0,tPen\WObj:=wPaper;
    MoveL Offs(pOrigin,266.15,316.31,0.00),v40,z0,tPen\WObj:=wPaper;
    MoveL Offs(pOrigin,266.15,316.31,0.00),v40,z0,tPen\WObj:=wPaper;
    MoveL Offs(pOrigin,266.79,317.09,0.00),v40,z0,tPen\WObj:=wPaper;
    MoveL Offs(pOrigin,268.91,317.38,0.00),v40,z0,tPen\WObj:=wPaper;
    MoveL Offs(pOrigin,268.91,317.38,0.00),v40,z0,tPen\WObj:=wPaper;
    MoveL Offs(pOrigin,269.55,318.30,0.00),v40,z0,tPen\WObj:=wPaper;
    MoveL Offs(pOrigin,273.38,320.56,0.00),v40,fine,tPen\WObj:=wPaper;
    MoveL Offs(pOrigin,273.38,320.56,6.00),v60,z5,tPen\WObj:=wPaper;
    MoveL Offs(pOrigin,275.71,318.23,6.00),vTravel,z5,tPen\WObj:=wPaper;
    MoveL Offs(pOrigin,275.71,318.23,0.00),v60,z0,tPen\WObj:=wPaper;
    MoveL Offs(pOrigin,272.95,316.88,0.00),v40,z0,tPen\WObj:=wPaper;
    MoveL Offs(pOrigin,271.25,316.52,0.00),v40,z0,tPen\WObj:=wPaper;
    MoveL Offs(pOrigin,271.25,316.52,0.00),v40,z0,tPen\WObj:=wPaper;
    MoveL Offs(pOrigin,270.40,315.46,0.00),v40,z0,tPen\WObj:=wPaper;
    MoveL Offs(pOrigin,269.34,315.25,0.00),v40,z0,tPen\WObj:=wPaper;
    MoveL Offs(pOrigin,269.34,315.25,0.00),v40,z0,tPen\WObj:=wPaper;
    MoveL Offs(pOrigin,268.13,313.76,0.00),v40,z0,tPen\WObj:=wPaper;
    MoveL Offs(pOrigin,270.40,313.34,0.00),v40,z0,tPen\WObj:=wPaper;
    MoveL Offs(pOrigin,271.04,312.91,0.00),v40,fine,tPen\WObj:=wPaper;
    MoveL Offs(pOrigin,271.04,312.91,6.00),v60,z5,tPen\WObj:=wPaper;
    MoveL Offs(pOrigin,270.61,311.64,6.00),vTravel,z5,tPen\WObj:=wPaper;
    MoveL Offs(pOrigin,270.61,311.64,0.00),v60,z0,tPen\WObj:=wPaper;
    MoveL Offs(pOrigin,268.49,311.85,0.00),v40,z0,tPen\WObj:=wPaper;
    MoveL Offs(pOrigin,267.42,311.42,0.00),v40,z0,tPen\WObj:=wPaper;
    MoveL Offs(pOrigin,265.94,311.42,0.00),v40,z0,tPen\WObj:=wPaper;
    MoveL Offs(pOrigin,260.84,309.73,0.00),v40,fine,tPen\WObj:=wPaper;
    MoveL Offs(pOrigin,260.84,309.73,6.00),v60,z5,tPen\WObj:=wPaper;
    MoveL Offs(pOrigin,258.08,310.36,6.00),vTravel,z5,tPen\WObj:=wPaper;
    MoveL Offs(pOrigin,258.08,310.36,0.00),v60,z0,tPen\WObj:=wPaper;
    MoveL Offs(pOrigin,259.35,311.50,0.00),v40,z0,tPen\WObj:=wPaper;
    MoveL Offs(pOrigin,261.69,312.70,0.00),v40,z0,tPen\WObj:=wPaper;
    MoveL Offs(pOrigin,263.17,313.12,0.00),v40,z0,tPen\WObj:=wPaper;
    MoveL Offs(pOrigin,268.06,313.55,0.00),v40,z0,tPen\WObj:=wPaper;
    MoveL Offs(pOrigin,267.42,313.34,0.00),v40,z0,tPen\WObj:=wPaper;
    MoveL Offs(pOrigin,267.64,312.27,0.00),v40,z0,tPen\WObj:=wPaper;
    MoveL Offs(pOrigin,268.06,311.85,0.00),v40,fine,tPen\WObj:=wPaper;
    MoveL Offs(pOrigin,268.06,311.85,6.00),v60,z5,tPen\WObj:=wPaper;
    MoveL Offs(pOrigin,269.34,315.25,6.00),vTravel,z5,tPen\WObj:=wPaper;
    MoveL Offs(pOrigin,269.34,315.25,0.00),v60,z0,tPen\WObj:=wPaper;
    MoveL Offs(pOrigin,267.21,315.46,0.00),v40,z0,tPen\WObj:=wPaper;
    MoveL Offs(pOrigin,266.15,316.31,0.00),v40,fine,tPen\WObj:=wPaper;
    MoveL Offs(pOrigin,266.15,316.31,6.00),v60,z5,tPen\WObj:=wPaper;
    MoveL Offs(pOrigin,264.02,316.10,6.00),vTravel,z5,tPen\WObj:=wPaper;
    MoveL Offs(pOrigin,264.02,316.10,0.00),v60,z0,tPen\WObj:=wPaper;
    MoveL Offs(pOrigin,263.60,315.60,0.00),v40,z0,tPen\WObj:=wPaper;
    MoveL Offs(pOrigin,259.14,314.05,0.00),v40,z0,tPen\WObj:=wPaper;
    MoveL Offs(pOrigin,257.86,313.12,0.00),v40,z0,tPen\WObj:=wPaper;
    MoveL Offs(pOrigin,256.16,311.21,0.00),v40,fine,tPen\WObj:=wPaper;
    MoveL Offs(pOrigin,256.16,311.21,6.00),v60,z5,tPen\WObj:=wPaper;
    MoveL Offs(pOrigin,253.82,311.21,6.00),vTravel,z5,tPen\WObj:=wPaper;
    MoveL Offs(pOrigin,253.82,311.21,0.00),v60,z0,tPen\WObj:=wPaper;
    MoveL Offs(pOrigin,254.25,313.34,0.00),v40,z0,tPen\WObj:=wPaper;
    MoveL Offs(pOrigin,254.25,313.34,0.00),v40,z0,tPen\WObj:=wPaper;
    MoveL Offs(pOrigin,253.40,313.12,0.00),v40,z0,tPen\WObj:=wPaper;
    MoveL Offs(pOrigin,252.76,311.64,0.00),v40,z0,tPen\WObj:=wPaper;
    MoveL Offs(pOrigin,252.12,312.49,0.00),v40,z0,tPen\WObj:=wPaper;
    MoveL Offs(pOrigin,252.55,313.76,0.00),v40,z0,tPen\WObj:=wPaper;
    MoveL Offs(pOrigin,252.34,315.04,0.00),v40,z0,tPen\WObj:=wPaper;
    MoveL Offs(pOrigin,252.34,315.04,0.00),v40,z0,tPen\WObj:=wPaper;
    MoveL Offs(pOrigin,252.98,316.31,0.00),v40,z0,tPen\WObj:=wPaper;
    MoveL Offs(pOrigin,252.98,316.31,0.00),v40,z0,tPen\WObj:=wPaper;
    MoveL Offs(pOrigin,254.04,316.74,0.00),v40,z0,tPen\WObj:=wPaper;
    MoveL Offs(pOrigin,254.53,318.01,0.00),v40,z0,tPen\WObj:=wPaper;
    MoveL Offs(pOrigin,255.52,318.44,0.00),v40,z0,tPen\WObj:=wPaper;
    MoveL Offs(pOrigin,255.95,318.01,0.00),v40,z0,tPen\WObj:=wPaper;
    MoveL Offs(pOrigin,259.56,320.56,0.00),v40,fine,tPen\WObj:=wPaper;
    MoveL Offs(pOrigin,259.56,320.56,6.00),v60,z5,tPen\WObj:=wPaper;
    MoveL Offs(pOrigin,260.20,321.62,6.00),vTravel,z5,tPen\WObj:=wPaper;
    MoveL Offs(pOrigin,260.20,321.62,0.00),v60,z0,tPen\WObj:=wPaper;
    MoveL Offs(pOrigin,261.05,322.48,0.00),v40,z0,tPen\WObj:=wPaper;
    MoveL Offs(pOrigin,260.20,321.62,0.00),v40,fine,tPen\WObj:=wPaper;
    MoveL Offs(pOrigin,260.20,321.62,6.00),v60,z5,tPen\WObj:=wPaper;
    MoveL Offs(pOrigin,261.26,322.69,6.00),vTravel,z5,tPen\WObj:=wPaper;
    MoveL Offs(pOrigin,261.26,322.69,0.00),v60,z0,tPen\WObj:=wPaper;
    MoveL Offs(pOrigin,261.90,323.33,0.00),v40,z0,tPen\WObj:=wPaper;
    MoveL Offs(pOrigin,261.26,322.69,0.00),v40,fine,tPen\WObj:=wPaper;
    MoveL Offs(pOrigin,261.26,322.69,6.00),v60,z5,tPen\WObj:=wPaper;
    MoveL Offs(pOrigin,262.54,324.39,6.00),vTravel,z5,tPen\WObj:=wPaper;
    MoveL Offs(pOrigin,262.54,324.39,0.00),v60,z0,tPen\WObj:=wPaper;
    MoveL Offs(pOrigin,262.75,324.81,0.00),v40,z0,tPen\WObj:=wPaper;
    MoveL Offs(pOrigin,262.54,324.39,0.00),v40,fine,tPen\WObj:=wPaper;
    MoveL Offs(pOrigin,262.54,324.39,6.00),v60,z5,tPen\WObj:=wPaper;
    MoveL Offs(pOrigin,266.15,325.45,6.00),vTravel,z5,tPen\WObj:=wPaper;
    MoveL Offs(pOrigin,266.15,325.45,0.00),v60,z0,tPen\WObj:=wPaper;
    MoveL Offs(pOrigin,266.36,325.88,0.00),v40,z0,tPen\WObj:=wPaper;
    MoveL Offs(pOrigin,266.15,325.45,0.00),v40,fine,tPen\WObj:=wPaper;
    MoveL Offs(pOrigin,266.15,325.45,6.00),v60,z5,tPen\WObj:=wPaper;
    MoveL Offs(pOrigin,267.85,324.81,6.00),vTravel,z5,tPen\WObj:=wPaper;
    MoveL Offs(pOrigin,267.85,324.81,0.00),v60,z0,tPen\WObj:=wPaper;
    MoveL Offs(pOrigin,268.06,325.24,0.00),v40,z0,tPen\WObj:=wPaper;
    MoveL Offs(pOrigin,267.85,324.81,0.00),v40,fine,tPen\WObj:=wPaper;
    MoveL Offs(pOrigin,267.85,324.81,6.00),v60,z5,tPen\WObj:=wPaper;
    MoveL Offs(pOrigin,271.89,326.51,6.00),vTravel,z5,tPen\WObj:=wPaper;
    MoveL Offs(pOrigin,271.89,326.51,0.00),v60,z0,tPen\WObj:=wPaper;
    MoveL Offs(pOrigin,269.34,324.17,0.00),v40,z0,tPen\WObj:=wPaper;
    MoveL Offs(pOrigin,267.85,321.84,0.00),v40,z0,tPen\WObj:=wPaper;
    MoveL Offs(pOrigin,266.36,320.56,0.00),v40,fine,tPen\WObj:=wPaper;
    MoveL Offs(pOrigin,266.36,320.56,6.00),v60,z5,tPen\WObj:=wPaper;
    MoveL Offs(pOrigin,268.06,320.14,6.00),vTravel,z5,tPen\WObj:=wPaper;
    MoveL Offs(pOrigin,268.06,320.14,0.00),v60,z0,tPen\WObj:=wPaper;
    MoveL Offs(pOrigin,268.49,320.35,0.00),v40,z0,tPen\WObj:=wPaper;
    MoveL Offs(pOrigin,268.06,320.14,0.00),v40,fine,tPen\WObj:=wPaper;
    MoveL Offs(pOrigin,268.06,320.14,6.00),v60,z5,tPen\WObj:=wPaper;
    MoveL Offs(pOrigin,268.91,317.38,6.00),vTravel,z5,tPen\WObj:=wPaper;
    MoveL Offs(pOrigin,268.91,317.38,0.00),v60,z0,tPen\WObj:=wPaper;
    MoveL Offs(pOrigin,271.04,317.45,0.00),v40,z0,tPen\WObj:=wPaper;
    MoveL Offs(pOrigin,273.38,318.58,0.00),v40,z0,tPen\WObj:=wPaper;
    MoveL Offs(pOrigin,276.77,320.85,0.00),v40,z0,tPen\WObj:=wPaper;
    MoveL Offs(pOrigin,279.11,321.84,0.00),v40,z0,tPen\WObj:=wPaper;
    MoveL Offs(pOrigin,283.72,322.05,0.00),v40,z0,tPen\WObj:=wPaper;
    MoveL Offs(pOrigin,283.50,323.04,0.00),v40,z0,tPen\WObj:=wPaper;
  ENDPROC

  PROC DrawPart28()
    MoveL Offs(pOrigin,281.88,324.03,0.00),v40,z0,tPen\WObj:=wPaper;
    MoveL Offs(pOrigin,280.60,324.39,0.00),v40,z0,tPen\WObj:=wPaper;
    MoveL Offs(pOrigin,279.33,323.75,0.00),v40,z0,tPen\WObj:=wPaper;
    MoveL Offs(pOrigin,280.17,324.39,0.00),v40,z0,tPen\WObj:=wPaper;
    MoveL Offs(pOrigin,279.96,324.81,0.00),v40,z0,tPen\WObj:=wPaper;
    MoveL Offs(pOrigin,278.90,325.02,0.00),v40,z0,tPen\WObj:=wPaper;
    MoveL Offs(pOrigin,275.71,324.81,0.00),v40,z0,tPen\WObj:=wPaper;
    MoveL Offs(pOrigin,272.74,323.61,0.00),v40,z0,tPen\WObj:=wPaper;
    MoveL Offs(pOrigin,267.42,319.64,0.00),v40,z0,tPen\WObj:=wPaper;
    MoveL Offs(pOrigin,263.81,318.86,0.00),v40,z0,tPen\WObj:=wPaper;
    MoveL Offs(pOrigin,263.39,319.08,0.00),v40,fine,tPen\WObj:=wPaper;
    MoveL Offs(pOrigin,263.39,319.08,6.00),v60,z5,tPen\WObj:=wPaper;
    MoveL Offs(pOrigin,259.35,316.95,6.00),vTravel,z5,tPen\WObj:=wPaper;
    MoveL Offs(pOrigin,259.35,316.95,0.00),v60,z0,tPen\WObj:=wPaper;
    MoveL Offs(pOrigin,256.38,315.46,0.00),v40,z0,tPen\WObj:=wPaper;
    MoveL Offs(pOrigin,254.25,313.34,0.00),v40,fine,tPen\WObj:=wPaper;
    MoveL Offs(pOrigin,254.25,313.34,6.00),v60,z5,tPen\WObj:=wPaper;
    MoveL Offs(pOrigin,252.34,315.04,6.00),vTravel,z5,tPen\WObj:=wPaper;
    MoveL Offs(pOrigin,252.34,315.04,0.00),v60,z0,tPen\WObj:=wPaper;
    MoveL Offs(pOrigin,251.42,314.40,0.00),v40,z0,tPen\WObj:=wPaper;
    MoveL Offs(pOrigin,251.06,311.85,0.00),v40,fine,tPen\WObj:=wPaper;
    MoveL Offs(pOrigin,251.06,311.85,6.00),v60,z5,tPen\WObj:=wPaper;
    MoveL Offs(pOrigin,249.57,312.06,6.00),vTravel,z5,tPen\WObj:=wPaper;
    MoveL Offs(pOrigin,249.57,312.06,0.00),v60,z0,tPen\WObj:=wPaper;
    MoveL Offs(pOrigin,249.15,313.76,0.00),v40,z0,tPen\WObj:=wPaper;
    MoveL Offs(pOrigin,249.86,315.89,0.00),v40,z0,tPen\WObj:=wPaper;
    MoveL Offs(pOrigin,251.49,318.01,0.00),v40,z0,tPen\WObj:=wPaper;
    MoveL Offs(pOrigin,252.76,318.44,0.00),v40,z0,tPen\WObj:=wPaper;
    MoveL Offs(pOrigin,252.76,318.44,0.00),v40,z0,tPen\WObj:=wPaper;
    MoveL Offs(pOrigin,256.16,321.20,0.00),v40,z0,tPen\WObj:=wPaper;
    MoveL Offs(pOrigin,257.01,322.69,0.00),v40,z0,tPen\WObj:=wPaper;
    MoveL Offs(pOrigin,257.01,322.69,0.00),v40,z0,tPen\WObj:=wPaper;
    MoveL Offs(pOrigin,258.08,323.96,0.00),v40,z0,tPen\WObj:=wPaper;
    MoveL Offs(pOrigin,258.08,323.96,0.00),v40,z0,tPen\WObj:=wPaper;
    MoveL Offs(pOrigin,259.28,324.60,0.00),v40,z0,tPen\WObj:=wPaper;
    MoveL Offs(pOrigin,260.20,326.73,0.00),v40,z0,tPen\WObj:=wPaper;
    MoveL Offs(pOrigin,260.41,329.91,0.00),v40,z0,tPen\WObj:=wPaper;
    MoveL Offs(pOrigin,260.20,331.19,0.00),v40,z0,tPen\WObj:=wPaper;
    MoveL Offs(pOrigin,259.63,332.46,0.00),v40,z0,tPen\WObj:=wPaper;
    MoveL Offs(pOrigin,258.36,333.31,0.00),v40,z0,tPen\WObj:=wPaper;
    MoveL Offs(pOrigin,256.16,336.22,0.00),v40,z0,tPen\WObj:=wPaper;
    MoveL Offs(pOrigin,254.25,337.35,0.00),v40,z0,tPen\WObj:=wPaper;
    MoveL Offs(pOrigin,253.75,338.41,0.00),v40,z0,tPen\WObj:=wPaper;
    MoveL Offs(pOrigin,254.89,338.62,0.00),v40,z0,tPen\WObj:=wPaper;
    MoveL Offs(pOrigin,259.14,336.92,0.00),v40,fine,tPen\WObj:=wPaper;
    MoveL Offs(pOrigin,259.14,336.92,6.00),v60,z5,tPen\WObj:=wPaper;
    MoveL Offs(pOrigin,260.84,334.80,6.00),vTravel,z5,tPen\WObj:=wPaper;
    MoveL Offs(pOrigin,260.84,334.80,0.00),v60,z0,tPen\WObj:=wPaper;
    MoveL Offs(pOrigin,260.62,335.23,0.00),v40,z0,tPen\WObj:=wPaper;
    MoveL Offs(pOrigin,260.84,334.80,0.00),v40,fine,tPen\WObj:=wPaper;
    MoveL Offs(pOrigin,260.84,334.80,6.00),v60,z5,tPen\WObj:=wPaper;
    MoveL Offs(pOrigin,258.29,333.10,6.00),vTravel,z5,tPen\WObj:=wPaper;
    MoveL Offs(pOrigin,258.29,333.10,0.00),v60,z0,tPen\WObj:=wPaper;
    MoveL Offs(pOrigin,258.71,330.55,0.00),v40,z0,tPen\WObj:=wPaper;
    MoveL Offs(pOrigin,258.71,327.36,0.00),v40,z0,tPen\WObj:=wPaper;
    MoveL Offs(pOrigin,258.08,325.24,0.00),v40,z0,tPen\WObj:=wPaper;
    MoveL Offs(pOrigin,258.08,323.96,0.00),v40,fine,tPen\WObj:=wPaper;
    MoveL Offs(pOrigin,258.08,323.96,6.00),v60,z5,tPen\WObj:=wPaper;
    MoveL Offs(pOrigin,257.01,322.69,6.00),vTravel,z5,tPen\WObj:=wPaper;
    MoveL Offs(pOrigin,257.01,322.69,0.00),v60,z0,tPen\WObj:=wPaper;
    MoveL Offs(pOrigin,256.38,322.90,0.00),v40,z0,tPen\WObj:=wPaper;
    MoveL Offs(pOrigin,254.89,322.05,0.00),v40,z0,tPen\WObj:=wPaper;
    MoveL Offs(pOrigin,254.04,322.26,0.00),v40,z0,tPen\WObj:=wPaper;
    MoveL Offs(pOrigin,254.04,322.26,0.00),v40,z0,tPen\WObj:=wPaper;
    MoveL Offs(pOrigin,255.81,325.45,0.00),v40,z0,tPen\WObj:=wPaper;
    MoveL Offs(pOrigin,256.16,327.36,0.00),v40,z0,tPen\WObj:=wPaper;
    MoveL Offs(pOrigin,255.95,329.49,0.00),v40,z0,tPen\WObj:=wPaper;
    MoveL Offs(pOrigin,255.38,331.19,0.00),v40,z0,tPen\WObj:=wPaper;
    MoveL Offs(pOrigin,253.82,333.52,0.00),v40,fine,tPen\WObj:=wPaper;
    MoveL Offs(pOrigin,253.82,333.52,6.00),v60,z5,tPen\WObj:=wPaper;
    MoveL Offs(pOrigin,254.04,336.29,6.00),vTravel,z5,tPen\WObj:=wPaper;
    MoveL Offs(pOrigin,254.04,336.29,0.00),v60,z0,tPen\WObj:=wPaper;
    MoveL Offs(pOrigin,256.45,333.10,0.00),v40,z0,tPen\WObj:=wPaper;
    MoveL Offs(pOrigin,256.80,332.04,0.00),v40,fine,tPen\WObj:=wPaper;
    MoveL Offs(pOrigin,256.80,332.04,6.00),v60,z5,tPen\WObj:=wPaper;
    MoveL Offs(pOrigin,252.34,330.98,6.00),vTravel,z5,tPen\WObj:=wPaper;
    MoveL Offs(pOrigin,252.34,330.98,0.00),v60,z0,tPen\WObj:=wPaper;
    MoveL Offs(pOrigin,252.12,331.40,0.00),v40,z0,tPen\WObj:=wPaper;
    MoveL Offs(pOrigin,252.34,330.98,0.00),v40,fine,tPen\WObj:=wPaper;
    MoveL Offs(pOrigin,252.34,330.98,6.00),v60,z5,tPen\WObj:=wPaper;
    MoveL Offs(pOrigin,249.79,331.83,6.00),vTravel,z5,tPen\WObj:=wPaper;
    MoveL Offs(pOrigin,249.79,331.83,0.00),v60,z0,tPen\WObj:=wPaper;
    MoveL Offs(pOrigin,249.57,332.25,0.00),v40,z0,tPen\WObj:=wPaper;
    MoveL Offs(pOrigin,249.79,331.83,0.00),v40,fine,tPen\WObj:=wPaper;
    MoveL Offs(pOrigin,249.79,331.83,6.00),v60,z5,tPen\WObj:=wPaper;
    MoveL Offs(pOrigin,247.02,330.98,6.00),vTravel,z5,tPen\WObj:=wPaper;
    MoveL Offs(pOrigin,247.02,330.98,0.00),v60,z0,tPen\WObj:=wPaper;
    MoveL Offs(pOrigin,246.46,332.46,0.00),v40,z0,tPen\WObj:=wPaper;
    MoveL Offs(pOrigin,244.05,335.23,0.00),v40,z0,tPen\WObj:=wPaper;
    MoveL Offs(pOrigin,242.99,335.65,0.00),v40,z0,tPen\WObj:=wPaper;
    MoveL Offs(pOrigin,242.63,335.44,0.00),v40,z0,tPen\WObj:=wPaper;
    MoveL Offs(pOrigin,242.85,334.59,0.00),v40,z0,tPen\WObj:=wPaper;
    MoveL Offs(pOrigin,244.33,332.67,0.00),v40,z0,tPen\WObj:=wPaper;
    MoveL Offs(pOrigin,244.69,331.61,0.00),v40,z0,tPen\WObj:=wPaper;
    MoveL Offs(pOrigin,244.90,328.64,0.00),v40,z0,tPen\WObj:=wPaper;
    MoveL Offs(pOrigin,243.70,325.66,0.00),v40,z0,tPen\WObj:=wPaper;
    MoveL Offs(pOrigin,242.07,323.54,0.00),v40,z0,tPen\WObj:=wPaper;
    MoveL Offs(pOrigin,242.35,323.11,0.00),v40,z0,tPen\WObj:=wPaper;
    MoveL Offs(pOrigin,244.69,323.75,0.00),v40,z0,tPen\WObj:=wPaper;
    MoveL Offs(pOrigin,245.75,324.81,0.00),v40,z0,tPen\WObj:=wPaper;
    MoveL Offs(pOrigin,246.67,326.51,0.00),v40,z0,tPen\WObj:=wPaper;
    MoveL Offs(pOrigin,247.24,328.85,0.00),v40,z0,tPen\WObj:=wPaper;
    MoveL Offs(pOrigin,247.02,330.98,0.00),v40,z0,tPen\WObj:=wPaper;
    MoveL Offs(pOrigin,246.60,331.83,0.00),v40,z0,tPen\WObj:=wPaper;
    MoveL Offs(pOrigin,246.39,332.25,0.00),v40,z0,tPen\WObj:=wPaper;
    MoveL Offs(pOrigin,246.60,331.83,0.00),v40,fine,tPen\WObj:=wPaper;
    MoveL Offs(pOrigin,246.60,331.83,6.00),v60,z5,tPen\WObj:=wPaper;
    MoveL Offs(pOrigin,248.51,334.80,6.00),vTravel,z5,tPen\WObj:=wPaper;
    MoveL Offs(pOrigin,248.51,334.80,0.00),v60,z0,tPen\WObj:=wPaper;
    MoveL Offs(pOrigin,246.39,336.15,0.00),v40,z0,tPen\WObj:=wPaper;
    MoveL Offs(pOrigin,241.93,338.13,0.00),v40,z0,tPen\WObj:=wPaper;
    MoveL Offs(pOrigin,241.29,339.05,0.00),v40,fine,tPen\WObj:=wPaper;
    MoveL Offs(pOrigin,241.29,339.05,6.00),v60,z5,tPen\WObj:=wPaper;
    MoveL Offs(pOrigin,242.56,335.65,6.00),vTravel,z5,tPen\WObj:=wPaper;
    MoveL Offs(pOrigin,242.56,335.65,0.00),v60,z0,tPen\WObj:=wPaper;
    MoveL Offs(pOrigin,240.86,336.78,0.00),v40,z0,tPen\WObj:=wPaper;
    MoveL Offs(pOrigin,236.82,338.27,0.00),v40,z0,tPen\WObj:=wPaper;
    MoveL Offs(pOrigin,232.57,338.62,0.00),v40,z0,tPen\WObj:=wPaper;
    MoveL Offs(pOrigin,231.51,339.48,0.00),v40,fine,tPen\WObj:=wPaper;
    MoveL Offs(pOrigin,231.51,339.48,6.00),v60,z5,tPen\WObj:=wPaper;
  ENDPROC

  PROC DrawPart29()
    MoveL Offs(pOrigin,232.36,335.44,6.00),vTravel,z5,tPen\WObj:=wPaper;
    MoveL Offs(pOrigin,232.36,335.44,0.00),v60,z0,tPen\WObj:=wPaper;
    MoveL Offs(pOrigin,233.00,334.38,0.00),v40,z0,tPen\WObj:=wPaper;
    MoveL Offs(pOrigin,235.34,332.89,0.00),v40,z0,tPen\WObj:=wPaper;
    MoveL Offs(pOrigin,235.76,332.67,0.00),v40,z0,tPen\WObj:=wPaper;
    MoveL Offs(pOrigin,237.11,330.55,0.00),v40,z0,tPen\WObj:=wPaper;
    MoveL Offs(pOrigin,237.46,327.58,0.00),v40,z0,tPen\WObj:=wPaper;
    MoveL Offs(pOrigin,236.68,325.45,0.00),v40,z0,tPen\WObj:=wPaper;
    MoveL Offs(pOrigin,234.27,322.05,0.00),v40,z0,tPen\WObj:=wPaper;
    MoveL Offs(pOrigin,234.27,322.05,0.00),v40,z0,tPen\WObj:=wPaper;
    MoveL Offs(pOrigin,234.70,321.62,0.00),v40,z0,tPen\WObj:=wPaper;
    MoveL Offs(pOrigin,236.40,321.84,0.00),v40,z0,tPen\WObj:=wPaper;
    MoveL Offs(pOrigin,236.40,321.84,0.00),v40,z0,tPen\WObj:=wPaper;
    MoveL Offs(pOrigin,236.40,321.41,0.00),v40,z0,tPen\WObj:=wPaper;
    MoveL Offs(pOrigin,235.34,320.14,0.00),v40,z0,tPen\WObj:=wPaper;
    MoveL Offs(pOrigin,235.34,320.14,0.00),v40,z0,tPen\WObj:=wPaper;
    MoveL Offs(pOrigin,235.27,319.29,0.00),v40,z0,tPen\WObj:=wPaper;
    MoveL Offs(pOrigin,233.78,317.16,0.00),v40,z0,tPen\WObj:=wPaper;
    MoveL Offs(pOrigin,233.00,315.04,0.00),v40,z0,tPen\WObj:=wPaper;
    MoveL Offs(pOrigin,233.00,313.12,0.00),v40,z0,tPen\WObj:=wPaper;
    MoveL Offs(pOrigin,233.85,310.58,0.00),v40,fine,tPen\WObj:=wPaper;
    MoveL Offs(pOrigin,233.85,310.58,6.00),v60,z5,tPen\WObj:=wPaper;
    MoveL Offs(pOrigin,232.15,310.58,6.00),vTravel,z5,tPen\WObj:=wPaper;
    MoveL Offs(pOrigin,232.15,310.58,0.00),v60,z0,tPen\WObj:=wPaper;
    MoveL Offs(pOrigin,231.09,313.34,0.00),v40,z0,tPen\WObj:=wPaper;
    MoveL Offs(pOrigin,230.88,316.10,0.00),v40,z0,tPen\WObj:=wPaper;
    MoveL Offs(pOrigin,230.88,316.10,0.00),v40,z0,tPen\WObj:=wPaper;
    MoveL Offs(pOrigin,229.81,315.89,0.00),v40,z0,tPen\WObj:=wPaper;
    MoveL Offs(pOrigin,229.81,315.89,0.00),v40,z0,tPen\WObj:=wPaper;
    MoveL Offs(pOrigin,229.81,313.98,0.00),v40,z0,tPen\WObj:=wPaper;
    MoveL Offs(pOrigin,230.66,311.42,0.00),v40,fine,tPen\WObj:=wPaper;
    MoveL Offs(pOrigin,230.66,311.42,6.00),v60,z5,tPen\WObj:=wPaper;
    MoveL Offs(pOrigin,229.39,311.00,6.00),vTravel,z5,tPen\WObj:=wPaper;
    MoveL Offs(pOrigin,229.39,311.00,0.00),v60,z0,tPen\WObj:=wPaper;
    MoveL Offs(pOrigin,228.11,313.76,0.00),v40,z0,tPen\WObj:=wPaper;
    MoveL Offs(pOrigin,228.11,315.89,0.00),v40,z0,tPen\WObj:=wPaper;
    MoveL Offs(pOrigin,229.18,317.16,0.00),v40,z0,tPen\WObj:=wPaper;
    MoveL Offs(pOrigin,229.18,317.16,0.00),v40,z0,tPen\WObj:=wPaper;
    MoveL Offs(pOrigin,228.96,319.29,0.00),v40,z0,tPen\WObj:=wPaper;
    MoveL Offs(pOrigin,228.96,319.29,0.00),v40,z0,tPen\WObj:=wPaper;
    MoveL Offs(pOrigin,227.48,318.44,0.00),v40,z0,tPen\WObj:=wPaper;
    MoveL Offs(pOrigin,226.41,316.10,0.00),v40,z0,tPen\WObj:=wPaper;
    MoveL Offs(pOrigin,226.41,316.10,0.00),v40,z0,tPen\WObj:=wPaper;
    MoveL Offs(pOrigin,226.41,313.76,0.00),v40,z0,tPen\WObj:=wPaper;
    MoveL Offs(pOrigin,226.06,312.91,0.00),v40,z0,tPen\WObj:=wPaper;
    MoveL Offs(pOrigin,226.84,311.21,0.00),v40,z0,tPen\WObj:=wPaper;
    MoveL Offs(pOrigin,228.11,310.15,0.00),v40,fine,tPen\WObj:=wPaper;
    MoveL Offs(pOrigin,228.11,310.15,6.00),v60,z5,tPen\WObj:=wPaper;
    MoveL Offs(pOrigin,225.14,310.36,6.00),vTravel,z5,tPen\WObj:=wPaper;
    MoveL Offs(pOrigin,225.14,310.36,0.00),v60,z0,tPen\WObj:=wPaper;
    MoveL Offs(pOrigin,223.01,311.92,0.00),v40,z0,tPen\WObj:=wPaper;
    MoveL Offs(pOrigin,222.38,312.06,0.00),v40,z0,tPen\WObj:=wPaper;
    MoveL Offs(pOrigin,222.38,312.06,0.00),v40,z0,tPen\WObj:=wPaper;
    MoveL Offs(pOrigin,222.16,316.10,0.00),v40,z0,tPen\WObj:=wPaper;
    MoveL Offs(pOrigin,222.16,316.10,0.00),v40,z0,tPen\WObj:=wPaper;
    MoveL Offs(pOrigin,223.01,316.95,0.00),v40,z0,tPen\WObj:=wPaper;
    MoveL Offs(pOrigin,223.01,317.38,0.00),v40,z0,tPen\WObj:=wPaper;
    MoveL Offs(pOrigin,223.86,318.01,0.00),v40,z0,tPen\WObj:=wPaper;
    MoveL Offs(pOrigin,224.29,318.01,0.00),v40,z0,tPen\WObj:=wPaper;
    MoveL Offs(pOrigin,227.55,322.69,0.00),v40,z0,tPen\WObj:=wPaper;
    MoveL Offs(pOrigin,228.11,325.88,0.00),v40,z0,tPen\WObj:=wPaper;
    MoveL Offs(pOrigin,227.05,328.00,0.00),v40,z0,tPen\WObj:=wPaper;
    MoveL Offs(pOrigin,225.14,329.42,0.00),v40,z0,tPen\WObj:=wPaper;
    MoveL Offs(pOrigin,223.86,329.70,0.00),v40,z0,tPen\WObj:=wPaper;
    MoveL Offs(pOrigin,223.86,329.70,0.00),v40,z0,tPen\WObj:=wPaper;
    MoveL Offs(pOrigin,223.93,329.06,0.00),v40,z0,tPen\WObj:=wPaper;
    MoveL Offs(pOrigin,225.21,327.36,0.00),v40,z0,tPen\WObj:=wPaper;
    MoveL Offs(pOrigin,225.56,326.30,0.00),v40,z0,tPen\WObj:=wPaper;
    MoveL Offs(pOrigin,225.35,323.33,0.00),v40,z0,tPen\WObj:=wPaper;
    MoveL Offs(pOrigin,223.65,319.29,0.00),v40,z0,tPen\WObj:=wPaper;
    MoveL Offs(pOrigin,223.86,318.23,0.00),v40,z0,tPen\WObj:=wPaper;
    MoveL Offs(pOrigin,224.71,318.65,0.00),v40,z0,tPen\WObj:=wPaper;
    MoveL Offs(pOrigin,224.29,318.01,0.00),v40,z0,tPen\WObj:=wPaper;
    MoveL Offs(pOrigin,224.71,317.59,0.00),v40,z0,tPen\WObj:=wPaper;
    MoveL Offs(pOrigin,224.71,316.10,0.00),v40,z0,tPen\WObj:=wPaper;
    MoveL Offs(pOrigin,225.14,315.89,0.00),v40,fine,tPen\WObj:=wPaper;
    MoveL Offs(pOrigin,225.14,315.89,6.00),v60,z5,tPen\WObj:=wPaper;
    MoveL Offs(pOrigin,226.41,316.10,6.00),vTravel,z5,tPen\WObj:=wPaper;
    MoveL Offs(pOrigin,226.41,316.10,0.00),v60,z0,tPen\WObj:=wPaper;
    MoveL Offs(pOrigin,225.56,316.03,0.00),v40,z0,tPen\WObj:=wPaper;
    MoveL Offs(pOrigin,225.14,315.46,0.00),v40,z0,tPen\WObj:=wPaper;
    MoveL Offs(pOrigin,225.42,313.55,0.00),v40,z0,tPen\WObj:=wPaper;
    MoveL Offs(pOrigin,225.99,313.34,0.00),v40,fine,tPen\WObj:=wPaper;
    MoveL Offs(pOrigin,225.99,313.34,6.00),v60,z5,tPen\WObj:=wPaper;
    MoveL Offs(pOrigin,222.59,311.85,6.00),vTravel,z5,tPen\WObj:=wPaper;
    MoveL Offs(pOrigin,222.59,311.85,0.00),v60,z0,tPen\WObj:=wPaper;
    MoveL Offs(pOrigin,222.59,311.42,0.00),v40,z0,tPen\WObj:=wPaper;
    MoveL Offs(pOrigin,222.16,311.42,0.00),v40,z0,tPen\WObj:=wPaper;
    MoveL Offs(pOrigin,221.95,312.06,0.00),v40,z0,tPen\WObj:=wPaper;
    MoveL Offs(pOrigin,222.59,311.85,0.00),v40,z0,tPen\WObj:=wPaper;
    MoveL Offs(pOrigin,222.59,311.42,0.00),v40,z0,tPen\WObj:=wPaper;
    MoveL Offs(pOrigin,222.16,311.42,0.00),v40,z0,tPen\WObj:=wPaper;
    MoveL Offs(pOrigin,221.95,312.06,0.00),v40,z0,tPen\WObj:=wPaper;
    MoveL Offs(pOrigin,222.59,311.85,0.00),v40,fine,tPen\WObj:=wPaper;
    MoveL Offs(pOrigin,222.59,311.85,6.00),v60,z5,tPen\WObj:=wPaper;
    MoveL Offs(pOrigin,222.16,313.12,6.00),vTravel,z5,tPen\WObj:=wPaper;
    MoveL Offs(pOrigin,222.16,313.12,0.00),v60,z0,tPen\WObj:=wPaper;
    MoveL Offs(pOrigin,220.68,313.27,0.00),v40,z0,tPen\WObj:=wPaper;
    MoveL Offs(pOrigin,218.76,314.61,0.00),v40,z0,tPen\WObj:=wPaper;
    MoveL Offs(pOrigin,218.34,314.40,0.00),v40,z0,tPen\WObj:=wPaper;
    MoveL Offs(pOrigin,218.76,315.04,0.00),v40,z0,tPen\WObj:=wPaper;
    MoveL Offs(pOrigin,218.76,316.95,0.00),v40,z0,tPen\WObj:=wPaper;
    MoveL Offs(pOrigin,218.76,316.95,0.00),v40,z0,tPen\WObj:=wPaper;
    MoveL Offs(pOrigin,220.04,318.86,0.00),v40,z0,tPen\WObj:=wPaper;
    MoveL Offs(pOrigin,220.04,318.86,0.00),v40,z0,tPen\WObj:=wPaper;
    MoveL Offs(pOrigin,220.89,322.05,0.00),v40,z0,tPen\WObj:=wPaper;
    MoveL Offs(pOrigin,220.68,324.39,0.00),v40,z0,tPen\WObj:=wPaper;
    MoveL Offs(pOrigin,219.82,326.09,0.00),v40,z0,tPen\WObj:=wPaper;
    MoveL Offs(pOrigin,217.49,328.42,0.00),v40,z0,tPen\WObj:=wPaper;
    MoveL Offs(pOrigin,217.49,328.42,0.00),v40,z0,tPen\WObj:=wPaper;
    MoveL Offs(pOrigin,218.55,328.64,0.00),v40,z0,tPen\WObj:=wPaper;
    MoveL Offs(pOrigin,220.46,327.93,0.00),v40,z0,tPen\WObj:=wPaper;
    MoveL Offs(pOrigin,221.74,327.15,0.00),v40,z0,tPen\WObj:=wPaper;
    MoveL Offs(pOrigin,222.87,325.88,0.00),v40,z0,tPen\WObj:=wPaper;
    MoveL Offs(pOrigin,223.44,324.17,0.00),v40,z0,tPen\WObj:=wPaper;
    MoveL Offs(pOrigin,223.44,322.48,0.00),v40,z0,tPen\WObj:=wPaper;
    MoveL Offs(pOrigin,222.80,320.99,0.00),v40,z0,tPen\WObj:=wPaper;
    MoveL Offs(pOrigin,221.95,320.35,0.00),v40,z0,tPen\WObj:=wPaper;
    MoveL Offs(pOrigin,221.95,320.35,0.00),v40,z0,tPen\WObj:=wPaper;
    MoveL Offs(pOrigin,221.74,319.50,0.00),v40,z0,tPen\WObj:=wPaper;
  ENDPROC

  PROC DrawPart30()
    MoveL Offs(pOrigin,220.89,318.86,0.00),v40,z0,tPen\WObj:=wPaper;
    MoveL Offs(pOrigin,220.89,318.86,0.00),v40,z0,tPen\WObj:=wPaper;
    MoveL Offs(pOrigin,220.96,316.95,0.00),v40,z0,tPen\WObj:=wPaper;
    MoveL Offs(pOrigin,222.16,316.10,0.00),v40,fine,tPen\WObj:=wPaper;
    MoveL Offs(pOrigin,222.16,316.10,6.00),v60,z5,tPen\WObj:=wPaper;
    MoveL Offs(pOrigin,220.89,318.86,6.00),vTravel,z5,tPen\WObj:=wPaper;
    MoveL Offs(pOrigin,220.89,318.86,0.00),v60,z0,tPen\WObj:=wPaper;
    MoveL Offs(pOrigin,220.89,319.08,0.00),v40,z0,tPen\WObj:=wPaper;
    MoveL Offs(pOrigin,220.04,318.86,0.00),v40,fine,tPen\WObj:=wPaper;
    MoveL Offs(pOrigin,220.04,318.86,6.00),v60,z5,tPen\WObj:=wPaper;
    MoveL Offs(pOrigin,221.74,319.92,6.00),vTravel,z5,tPen\WObj:=wPaper;
    MoveL Offs(pOrigin,221.74,319.92,0.00),v60,z0,tPen\WObj:=wPaper;
    MoveL Offs(pOrigin,221.95,320.35,0.00),v40,z0,tPen\WObj:=wPaper;
    MoveL Offs(pOrigin,221.74,319.92,0.00),v40,z0,tPen\WObj:=wPaper;
    MoveL Offs(pOrigin,221.95,320.35,0.00),v40,z0,tPen\WObj:=wPaper;
    MoveL Offs(pOrigin,221.74,320.99,0.00),v40,z0,tPen\WObj:=wPaper;
    MoveL Offs(pOrigin,222.38,323.33,0.00),v40,fine,tPen\WObj:=wPaper;
    MoveL Offs(pOrigin,222.38,323.33,6.00),v60,z5,tPen\WObj:=wPaper;
    MoveL Offs(pOrigin,225.35,319.50,6.00),vTravel,z5,tPen\WObj:=wPaper;
    MoveL Offs(pOrigin,225.35,319.50,0.00),v60,z0,tPen\WObj:=wPaper;
    MoveL Offs(pOrigin,225.99,320.35,0.00),v40,z0,tPen\WObj:=wPaper;
    MoveL Offs(pOrigin,225.35,319.50,0.00),v40,fine,tPen\WObj:=wPaper;
    MoveL Offs(pOrigin,225.35,319.50,6.00),v60,z5,tPen\WObj:=wPaper;
    MoveL Offs(pOrigin,226.84,317.59,6.00),vTravel,z5,tPen\WObj:=wPaper;
    MoveL Offs(pOrigin,226.84,317.59,0.00),v60,z0,tPen\WObj:=wPaper;
    MoveL Offs(pOrigin,227.05,318.01,0.00),v40,z0,tPen\WObj:=wPaper;
    MoveL Offs(pOrigin,226.84,317.59,0.00),v40,fine,tPen\WObj:=wPaper;
    MoveL Offs(pOrigin,226.84,317.59,6.00),v60,z5,tPen\WObj:=wPaper;
    MoveL Offs(pOrigin,229.18,317.16,6.00),vTravel,z5,tPen\WObj:=wPaper;
    MoveL Offs(pOrigin,229.18,317.16,0.00),v60,z0,tPen\WObj:=wPaper;
    MoveL Offs(pOrigin,229.81,315.89,0.00),v40,z0,tPen\WObj:=wPaper;
    MoveL Offs(pOrigin,230.88,316.10,0.00),v40,z0,tPen\WObj:=wPaper;
    MoveL Offs(pOrigin,232.15,318.86,0.00),v40,z0,tPen\WObj:=wPaper;
    MoveL Offs(pOrigin,232.79,319.08,0.00),v40,z0,tPen\WObj:=wPaper;
    MoveL Offs(pOrigin,234.27,320.07,0.00),v40,z0,tPen\WObj:=wPaper;
    MoveL Offs(pOrigin,235.34,320.14,0.00),v40,fine,tPen\WObj:=wPaper;
    MoveL Offs(pOrigin,235.34,320.14,6.00),v60,z5,tPen\WObj:=wPaper;
    MoveL Offs(pOrigin,236.40,321.84,6.00),vTravel,z5,tPen\WObj:=wPaper;
    MoveL Offs(pOrigin,236.40,321.84,0.00),v60,z0,tPen\WObj:=wPaper;
    MoveL Offs(pOrigin,238.52,323.96,0.00),v40,z0,tPen\WObj:=wPaper;
    MoveL Offs(pOrigin,239.59,325.88,0.00),v40,z0,tPen\WObj:=wPaper;
    MoveL Offs(pOrigin,239.59,325.88,0.00),v40,z0,tPen\WObj:=wPaper;
    MoveL Offs(pOrigin,240.23,326.09,0.00),v40,z0,tPen\WObj:=wPaper;
    MoveL Offs(pOrigin,240.86,327.15,0.00),v40,z0,tPen\WObj:=wPaper;
    MoveL Offs(pOrigin,241.07,329.70,0.00),v40,z0,tPen\WObj:=wPaper;
    MoveL Offs(pOrigin,239.73,333.10,0.00),v40,z0,tPen\WObj:=wPaper;
    MoveL Offs(pOrigin,238.52,334.02,0.00),v40,z0,tPen\WObj:=wPaper;
    MoveL Offs(pOrigin,237.25,334.38,0.00),v40,z0,tPen\WObj:=wPaper;
    MoveL Offs(pOrigin,237.25,334.38,0.00),v40,z0,tPen\WObj:=wPaper;
    MoveL Offs(pOrigin,233.64,335.65,0.00),v40,z0,tPen\WObj:=wPaper;
    MoveL Offs(pOrigin,223.23,335.44,0.00),v40,z0,tPen\WObj:=wPaper;
    MoveL Offs(pOrigin,222.16,334.80,0.00),v40,z0,tPen\WObj:=wPaper;
    MoveL Offs(pOrigin,218.12,334.59,0.00),v40,z0,tPen\WObj:=wPaper;
    MoveL Offs(pOrigin,217.49,335.01,0.00),v40,fine,tPen\WObj:=wPaper;
    MoveL Offs(pOrigin,217.49,335.01,6.00),v60,z5,tPen\WObj:=wPaper;
    MoveL Offs(pOrigin,214.94,332.67,6.00),vTravel,z5,tPen\WObj:=wPaper;
    MoveL Offs(pOrigin,214.94,332.67,0.00),v60,z0,tPen\WObj:=wPaper;
    MoveL Offs(pOrigin,213.88,333.31,0.00),v40,z0,tPen\WObj:=wPaper;
    MoveL Offs(pOrigin,212.39,333.10,0.00),v40,z0,tPen\WObj:=wPaper;
    MoveL Offs(pOrigin,211.75,333.52,0.00),v40,z0,tPen\WObj:=wPaper;
    MoveL Offs(pOrigin,211.75,333.52,0.00),v40,z0,tPen\WObj:=wPaper;
    MoveL Offs(pOrigin,212.18,334.23,0.00),v40,z0,tPen\WObj:=wPaper;
    MoveL Offs(pOrigin,217.06,335.01,0.00),v40,z0,tPen\WObj:=wPaper;
    MoveL Offs(pOrigin,218.12,335.93,0.00),v40,z0,tPen\WObj:=wPaper;
    MoveL Offs(pOrigin,224.71,337.85,0.00),v40,z0,tPen\WObj:=wPaper;
    MoveL Offs(pOrigin,225.77,338.62,0.00),v40,z0,tPen\WObj:=wPaper;
    MoveL Offs(pOrigin,228.96,339.26,0.00),v40,z0,tPen\WObj:=wPaper;
    MoveL Offs(pOrigin,230.66,339.26,0.00),v40,z0,tPen\WObj:=wPaper;
    MoveL Offs(pOrigin,231.73,339.69,0.00),v40,z0,tPen\WObj:=wPaper;
    MoveL Offs(pOrigin,236.82,339.69,0.00),v40,z0,tPen\WObj:=wPaper;
    MoveL Offs(pOrigin,240.23,339.05,0.00),v40,z0,tPen\WObj:=wPaper;
    MoveL Offs(pOrigin,242.77,339.48,0.00),v40,z0,tPen\WObj:=wPaper;
    MoveL Offs(pOrigin,249.57,338.84,0.00),v40,z0,tPen\WObj:=wPaper;
    MoveL Offs(pOrigin,249.57,338.84,0.00),v40,z0,tPen\WObj:=wPaper;
    MoveL Offs(pOrigin,250.00,337.63,0.00),v40,z0,tPen\WObj:=wPaper;
    MoveL Offs(pOrigin,254.04,336.29,0.00),v40,fine,tPen\WObj:=wPaper;
    MoveL Offs(pOrigin,254.04,336.29,6.00),v60,z5,tPen\WObj:=wPaper;
    MoveL Offs(pOrigin,253.61,338.62,6.00),vTravel,z5,tPen\WObj:=wPaper;
    MoveL Offs(pOrigin,253.61,338.62,0.00),v60,z0,tPen\WObj:=wPaper;
    MoveL Offs(pOrigin,251.06,339.05,0.00),v40,z0,tPen\WObj:=wPaper;
    MoveL Offs(pOrigin,249.57,338.84,0.00),v40,fine,tPen\WObj:=wPaper;
    MoveL Offs(pOrigin,249.57,338.84,6.00),v60,z5,tPen\WObj:=wPaper;
    MoveL Offs(pOrigin,240.23,331.83,6.00),vTravel,z5,tPen\WObj:=wPaper;
    MoveL Offs(pOrigin,240.23,331.83,0.00),v60,z0,tPen\WObj:=wPaper;
    MoveL Offs(pOrigin,240.01,332.25,0.00),v40,z0,tPen\WObj:=wPaper;
    MoveL Offs(pOrigin,240.23,331.83,0.00),v40,fine,tPen\WObj:=wPaper;
    MoveL Offs(pOrigin,240.23,331.83,6.00),v60,z5,tPen\WObj:=wPaper;
    MoveL Offs(pOrigin,237.25,334.38,6.00),vTravel,z5,tPen\WObj:=wPaper;
    MoveL Offs(pOrigin,237.25,334.38,0.00),v60,z0,tPen\WObj:=wPaper;
    MoveL Offs(pOrigin,239.59,330.55,0.00),v40,z0,tPen\WObj:=wPaper;
    MoveL Offs(pOrigin,239.80,329.70,0.00),v40,z0,tPen\WObj:=wPaper;
    MoveL Offs(pOrigin,239.38,326.51,0.00),v40,z0,tPen\WObj:=wPaper;
    MoveL Offs(pOrigin,239.59,325.88,0.00),v40,fine,tPen\WObj:=wPaper;
    MoveL Offs(pOrigin,239.59,325.88,6.00),v60,z5,tPen\WObj:=wPaper;
    MoveL Offs(pOrigin,241.93,323.11,6.00),vTravel,z5,tPen\WObj:=wPaper;
    MoveL Offs(pOrigin,241.93,323.11,0.00),v60,z0,tPen\WObj:=wPaper;
    MoveL Offs(pOrigin,238.31,319.92,0.00),v40,z0,tPen\WObj:=wPaper;
    MoveL Offs(pOrigin,237.46,318.01,0.00),v40,z0,tPen\WObj:=wPaper;
    MoveL Offs(pOrigin,237.46,318.01,0.00),v40,z0,tPen\WObj:=wPaper;
    MoveL Offs(pOrigin,236.82,313.55,0.00),v40,z0,tPen\WObj:=wPaper;
    MoveL Offs(pOrigin,238.10,310.36,0.00),v40,fine,tPen\WObj:=wPaper;
    MoveL Offs(pOrigin,238.10,310.36,6.00),v60,z5,tPen\WObj:=wPaper;
    MoveL Offs(pOrigin,236.82,309.73,6.00),vTravel,z5,tPen\WObj:=wPaper;
    MoveL Offs(pOrigin,236.82,309.73,0.00),v60,z0,tPen\WObj:=wPaper;
    MoveL Offs(pOrigin,235.69,311.00,0.00),v40,z0,tPen\WObj:=wPaper;
    MoveL Offs(pOrigin,235.12,312.70,0.00),v40,z0,tPen\WObj:=wPaper;
    MoveL Offs(pOrigin,235.12,315.04,0.00),v40,z0,tPen\WObj:=wPaper;
    MoveL Offs(pOrigin,236.19,317.38,0.00),v40,z0,tPen\WObj:=wPaper;
    MoveL Offs(pOrigin,237.46,318.01,0.00),v40,z0,tPen\WObj:=wPaper;
    MoveL Offs(pOrigin,236.40,317.80,0.00),v40,z0,tPen\WObj:=wPaper;
    MoveL Offs(pOrigin,236.82,318.01,0.00),v40,z0,tPen\WObj:=wPaper;
    MoveL Offs(pOrigin,236.40,317.80,0.00),v40,fine,tPen\WObj:=wPaper;
    MoveL Offs(pOrigin,236.40,317.80,6.00),v60,z5,tPen\WObj:=wPaper;
    MoveL Offs(pOrigin,235.55,316.52,6.00),vTravel,z5,tPen\WObj:=wPaper;
    MoveL Offs(pOrigin,235.55,316.52,0.00),v60,z0,tPen\WObj:=wPaper;
    MoveL Offs(pOrigin,235.76,316.95,0.00),v40,z0,tPen\WObj:=wPaper;
    MoveL Offs(pOrigin,235.55,316.52,0.00),v40,fine,tPen\WObj:=wPaper;
    MoveL Offs(pOrigin,235.55,316.52,6.00),v60,z5,tPen\WObj:=wPaper;
    MoveL Offs(pOrigin,239.16,316.10,6.00),vTravel,z5,tPen\WObj:=wPaper;
    MoveL Offs(pOrigin,239.16,316.10,0.00),v60,z0,tPen\WObj:=wPaper;
  ENDPROC

  PROC DrawPart31()
    MoveL Offs(pOrigin,239.38,316.52,0.00),v40,z0,tPen\WObj:=wPaper;
    MoveL Offs(pOrigin,239.16,316.10,0.00),v40,fine,tPen\WObj:=wPaper;
    MoveL Offs(pOrigin,239.16,316.10,6.00),v60,z5,tPen\WObj:=wPaper;
    MoveL Offs(pOrigin,240.44,318.44,6.00),vTravel,z5,tPen\WObj:=wPaper;
    MoveL Offs(pOrigin,240.44,318.44,0.00),v60,z0,tPen\WObj:=wPaper;
    MoveL Offs(pOrigin,240.86,318.86,0.00),v40,z0,tPen\WObj:=wPaper;
    MoveL Offs(pOrigin,240.44,318.44,0.00),v40,fine,tPen\WObj:=wPaper;
    MoveL Offs(pOrigin,240.44,318.44,6.00),v60,z5,tPen\WObj:=wPaper;
    MoveL Offs(pOrigin,242.14,319.71,6.00),vTravel,z5,tPen\WObj:=wPaper;
    MoveL Offs(pOrigin,242.14,319.71,0.00),v60,z0,tPen\WObj:=wPaper;
    MoveL Offs(pOrigin,242.56,319.08,0.00),v40,z0,tPen\WObj:=wPaper;
    MoveL Offs(pOrigin,241.93,317.38,0.00),v40,z0,tPen\WObj:=wPaper;
    MoveL Offs(pOrigin,242.14,316.60,0.00),v40,z0,tPen\WObj:=wPaper;
    MoveL Offs(pOrigin,242.77,316.95,0.00),v40,z0,tPen\WObj:=wPaper;
    MoveL Offs(pOrigin,244.05,318.65,0.00),v40,z0,tPen\WObj:=wPaper;
    MoveL Offs(pOrigin,245.96,319.29,0.00),v40,z0,tPen\WObj:=wPaper;
    MoveL Offs(pOrigin,245.96,319.29,0.00),v40,z0,tPen\WObj:=wPaper;
    MoveL Offs(pOrigin,250.21,322.69,0.00),v40,fine,tPen\WObj:=wPaper;
    MoveL Offs(pOrigin,250.21,322.69,6.00),v60,z5,tPen\WObj:=wPaper;
    MoveL Offs(pOrigin,251.27,325.24,6.00),vTravel,z5,tPen\WObj:=wPaper;
    MoveL Offs(pOrigin,251.27,325.24,0.00),v60,z0,tPen\WObj:=wPaper;
    MoveL Offs(pOrigin,250.28,323.54,0.00),v40,z0,tPen\WObj:=wPaper;
    MoveL Offs(pOrigin,250.43,322.76,0.00),v40,z0,tPen\WObj:=wPaper;
    MoveL Offs(pOrigin,251.49,323.33,0.00),v40,z0,tPen\WObj:=wPaper;
    MoveL Offs(pOrigin,252.83,325.66,0.00),v40,z0,tPen\WObj:=wPaper;
    MoveL Offs(pOrigin,253.19,326.94,0.00),v40,z0,tPen\WObj:=wPaper;
    MoveL Offs(pOrigin,252.98,329.49,0.00),v40,z0,tPen\WObj:=wPaper;
    MoveL Offs(pOrigin,252.41,331.19,0.00),v40,z0,tPen\WObj:=wPaper;
    MoveL Offs(pOrigin,251.27,332.89,0.00),v40,z0,tPen\WObj:=wPaper;
    MoveL Offs(pOrigin,249.57,334.52,0.00),v40,z0,tPen\WObj:=wPaper;
    MoveL Offs(pOrigin,248.73,334.73,0.00),v40,z0,tPen\WObj:=wPaper;
    MoveL Offs(pOrigin,248.58,333.95,0.00),v40,z0,tPen\WObj:=wPaper;
    MoveL Offs(pOrigin,249.86,332.04,0.00),v40,z0,tPen\WObj:=wPaper;
    MoveL Offs(pOrigin,250.43,329.91,0.00),v40,z0,tPen\WObj:=wPaper;
    MoveL Offs(pOrigin,250.43,328.64,0.00),v40,z0,tPen\WObj:=wPaper;
    MoveL Offs(pOrigin,249.65,325.88,0.00),v40,z0,tPen\WObj:=wPaper;
    MoveL Offs(pOrigin,248.30,323.61,0.00),v40,z0,tPen\WObj:=wPaper;
    MoveL Offs(pOrigin,243.62,320.28,0.00),v40,z0,tPen\WObj:=wPaper;
    MoveL Offs(pOrigin,242.77,320.14,0.00),v40,z0,tPen\WObj:=wPaper;
    MoveL Offs(pOrigin,242.77,320.14,0.00),v40,z0,tPen\WObj:=wPaper;
    MoveL Offs(pOrigin,242.42,320.99,0.00),v40,z0,tPen\WObj:=wPaper;
    MoveL Offs(pOrigin,243.84,322.26,0.00),v40,z0,tPen\WObj:=wPaper;
    MoveL Offs(pOrigin,244.48,323.54,0.00),v40,fine,tPen\WObj:=wPaper;
    MoveL Offs(pOrigin,244.48,323.54,6.00),v60,z5,tPen\WObj:=wPaper;
    MoveL Offs(pOrigin,246.60,322.48,6.00),vTravel,z5,tPen\WObj:=wPaper;
    MoveL Offs(pOrigin,246.60,322.48,0.00),v60,z0,tPen\WObj:=wPaper;
    MoveL Offs(pOrigin,247.45,323.33,0.00),v40,z0,tPen\WObj:=wPaper;
    MoveL Offs(pOrigin,247.45,323.33,0.00),v40,z0,tPen\WObj:=wPaper;
    MoveL Offs(pOrigin,247.88,324.81,0.00),v40,z0,tPen\WObj:=wPaper;
    MoveL Offs(pOrigin,247.66,324.39,0.00),v40,z0,tPen\WObj:=wPaper;
    MoveL Offs(pOrigin,247.88,324.81,0.00),v40,z0,tPen\WObj:=wPaper;
    MoveL Offs(pOrigin,247.66,324.39,0.00),v40,fine,tPen\WObj:=wPaper;
    MoveL Offs(pOrigin,247.66,324.39,6.00),v60,z5,tPen\WObj:=wPaper;
    MoveL Offs(pOrigin,246.39,325.66,6.00),vTravel,z5,tPen\WObj:=wPaper;
    MoveL Offs(pOrigin,246.39,325.66,0.00),v60,z0,tPen\WObj:=wPaper;
    MoveL Offs(pOrigin,246.60,326.09,0.00),v40,z0,tPen\WObj:=wPaper;
    MoveL Offs(pOrigin,246.39,325.66,0.00),v40,fine,tPen\WObj:=wPaper;
    MoveL Offs(pOrigin,246.39,325.66,6.00),v60,z5,tPen\WObj:=wPaper;
    MoveL Offs(pOrigin,242.99,321.62,6.00),vTravel,z5,tPen\WObj:=wPaper;
    MoveL Offs(pOrigin,242.99,321.62,0.00),v60,z0,tPen\WObj:=wPaper;
    MoveL Offs(pOrigin,243.84,322.48,0.00),v40,z0,tPen\WObj:=wPaper;
    MoveL Offs(pOrigin,242.99,321.62,0.00),v40,fine,tPen\WObj:=wPaper;
    MoveL Offs(pOrigin,242.99,321.62,6.00),v60,z5,tPen\WObj:=wPaper;
    MoveL Offs(pOrigin,242.14,319.71,6.00),vTravel,z5,tPen\WObj:=wPaper;
    MoveL Offs(pOrigin,242.14,319.71,0.00),v60,z0,tPen\WObj:=wPaper;
    MoveL Offs(pOrigin,241.15,319.08,0.00),v40,z0,tPen\WObj:=wPaper;
    MoveL Offs(pOrigin,240.01,317.59,0.00),v40,z0,tPen\WObj:=wPaper;
    MoveL Offs(pOrigin,238.95,315.04,0.00),v40,z0,tPen\WObj:=wPaper;
    MoveL Offs(pOrigin,238.95,312.70,0.00),v40,z0,tPen\WObj:=wPaper;
    MoveL Offs(pOrigin,240.23,310.15,0.00),v40,fine,tPen\WObj:=wPaper;
    MoveL Offs(pOrigin,240.23,310.15,6.00),v60,z5,tPen\WObj:=wPaper;
    MoveL Offs(pOrigin,241.50,311.64,6.00),vTravel,z5,tPen\WObj:=wPaper;
    MoveL Offs(pOrigin,241.50,311.64,0.00),v60,z0,tPen\WObj:=wPaper;
    MoveL Offs(pOrigin,241.29,312.49,0.00),v40,z0,tPen\WObj:=wPaper;
    MoveL Offs(pOrigin,241.71,312.91,0.00),v40,z0,tPen\WObj:=wPaper;
    MoveL Offs(pOrigin,241.71,312.91,0.00),v40,z0,tPen\WObj:=wPaper;
    MoveL Offs(pOrigin,241.50,314.40,0.00),v40,z0,tPen\WObj:=wPaper;
    MoveL Offs(pOrigin,241.93,316.52,0.00),v40,z0,tPen\WObj:=wPaper;
    MoveL Offs(pOrigin,242.99,316.95,0.00),v40,z0,tPen\WObj:=wPaper;
    MoveL Offs(pOrigin,243.41,317.59,0.00),v40,z0,tPen\WObj:=wPaper;
    MoveL Offs(pOrigin,242.99,316.95,0.00),v40,fine,tPen\WObj:=wPaper;
    MoveL Offs(pOrigin,242.99,316.95,6.00),v60,z5,tPen\WObj:=wPaper;
    MoveL Offs(pOrigin,245.96,318.44,6.00),vTravel,z5,tPen\WObj:=wPaper;
    MoveL Offs(pOrigin,245.96,318.44,0.00),v60,z0,tPen\WObj:=wPaper;
    MoveL Offs(pOrigin,244.48,315.04,0.00),v40,z0,tPen\WObj:=wPaper;
    MoveL Offs(pOrigin,244.48,312.91,0.00),v40,z0,tPen\WObj:=wPaper;
    MoveL Offs(pOrigin,245.32,311.00,0.00),v40,fine,tPen\WObj:=wPaper;
    MoveL Offs(pOrigin,245.32,311.00,6.00),v60,z5,tPen\WObj:=wPaper;
    MoveL Offs(pOrigin,247.02,311.85,6.00),vTravel,z5,tPen\WObj:=wPaper;
    MoveL Offs(pOrigin,247.02,311.85,0.00),v60,z0,tPen\WObj:=wPaper;
    MoveL Offs(pOrigin,246.81,314.19,0.00),v40,z0,tPen\WObj:=wPaper;
    MoveL Offs(pOrigin,247.31,315.89,0.00),v40,z0,tPen\WObj:=wPaper;
    MoveL Offs(pOrigin,249.36,318.44,0.00),v40,z0,tPen\WObj:=wPaper;
    MoveL Offs(pOrigin,249.79,319.50,0.00),v40,z0,tPen\WObj:=wPaper;
    MoveL Offs(pOrigin,249.79,319.50,0.00),v40,z0,tPen\WObj:=wPaper;
    MoveL Offs(pOrigin,246.81,318.44,0.00),v40,z0,tPen\WObj:=wPaper;
    MoveL Offs(pOrigin,246.03,318.65,0.00),v40,z0,tPen\WObj:=wPaper;
    MoveL Offs(pOrigin,245.96,319.29,0.00),v40,fine,tPen\WObj:=wPaper;
    MoveL Offs(pOrigin,245.96,319.29,6.00),v60,z5,tPen\WObj:=wPaper;
    MoveL Offs(pOrigin,249.79,319.50,6.00),vTravel,z5,tPen\WObj:=wPaper;
    MoveL Offs(pOrigin,249.79,319.50,0.00),v60,z0,tPen\WObj:=wPaper;
    MoveL Offs(pOrigin,254.04,322.26,0.00),v40,fine,tPen\WObj:=wPaper;
    MoveL Offs(pOrigin,254.04,322.26,6.00),v60,z5,tPen\WObj:=wPaper;
    MoveL Offs(pOrigin,252.76,318.44,6.00),vTravel,z5,tPen\WObj:=wPaper;
    MoveL Offs(pOrigin,252.76,318.44,0.00),v60,z0,tPen\WObj:=wPaper;
    MoveL Offs(pOrigin,252.76,317.16,0.00),v40,z0,tPen\WObj:=wPaper;
    MoveL Offs(pOrigin,252.76,316.95,0.00),v40,z0,tPen\WObj:=wPaper;
    MoveL Offs(pOrigin,252.98,316.74,0.00),v40,z0,tPen\WObj:=wPaper;
    MoveL Offs(pOrigin,253.19,316.95,0.00),v40,z0,tPen\WObj:=wPaper;
    MoveL Offs(pOrigin,252.98,317.16,0.00),v40,z0,tPen\WObj:=wPaper;
    MoveL Offs(pOrigin,252.76,316.95,0.00),v40,z0,tPen\WObj:=wPaper;
    MoveL Offs(pOrigin,252.98,316.74,0.00),v40,z0,tPen\WObj:=wPaper;
    MoveL Offs(pOrigin,253.19,316.95,0.00),v40,z0,tPen\WObj:=wPaper;
    MoveL Offs(pOrigin,252.98,317.16,0.00),v40,z0,tPen\WObj:=wPaper;
    MoveL Offs(pOrigin,252.76,316.95,0.00),v40,z0,tPen\WObj:=wPaper;
    MoveL Offs(pOrigin,252.76,315.89,0.00),v40,z0,tPen\WObj:=wPaper;
    MoveL Offs(pOrigin,252.98,316.31,0.00),v40,z0,tPen\WObj:=wPaper;
    MoveL Offs(pOrigin,252.76,315.89,0.00),v40,fine,tPen\WObj:=wPaper;
    MoveL Offs(pOrigin,252.76,315.89,6.00),v60,z5,tPen\WObj:=wPaper;
    MoveL Offs(pOrigin,254.25,316.74,6.00),vTravel,z5,tPen\WObj:=wPaper;
  ENDPROC

  PROC DrawPart32()
    MoveL Offs(pOrigin,254.25,316.74,0.00),v60,z0,tPen\WObj:=wPaper;
    MoveL Offs(pOrigin,255.31,316.95,0.00),v40,z0,tPen\WObj:=wPaper;
    MoveL Offs(pOrigin,255.95,317.59,0.00),v40,z0,tPen\WObj:=wPaper;
    MoveL Offs(pOrigin,255.95,318.01,0.00),v40,fine,tPen\WObj:=wPaper;
    MoveL Offs(pOrigin,255.95,318.01,6.00),v60,z5,tPen\WObj:=wPaper;
    MoveL Offs(pOrigin,257.23,319.29,6.00),vTravel,z5,tPen\WObj:=wPaper;
    MoveL Offs(pOrigin,257.23,319.29,0.00),v60,z0,tPen\WObj:=wPaper;
    MoveL Offs(pOrigin,257.65,319.50,0.00),v40,z0,tPen\WObj:=wPaper;
    MoveL Offs(pOrigin,257.23,319.29,0.00),v40,fine,tPen\WObj:=wPaper;
    MoveL Offs(pOrigin,257.23,319.29,6.00),v60,z5,tPen\WObj:=wPaper;
    MoveL Offs(pOrigin,264.88,308.66,6.00),vTravel,z5,tPen\WObj:=wPaper;
    MoveL Offs(pOrigin,264.88,308.66,0.00),v60,z0,tPen\WObj:=wPaper;
    MoveL Offs(pOrigin,267.00,309.30,0.00),v40,z0,tPen\WObj:=wPaper;
    MoveL Offs(pOrigin,271.89,308.88,0.00),v40,z0,tPen\WObj:=wPaper;
    MoveL Offs(pOrigin,274.01,308.02,0.00),v40,z0,tPen\WObj:=wPaper;
    MoveL Offs(pOrigin,274.01,308.02,0.00),v40,z0,tPen\WObj:=wPaper;
    MoveL Offs(pOrigin,276.77,308.24,0.00),v40,z0,tPen\WObj:=wPaper;
    MoveL Offs(pOrigin,277.84,309.09,0.00),v40,z0,tPen\WObj:=wPaper;
    MoveL Offs(pOrigin,280.60,309.94,0.00),v40,z0,tPen\WObj:=wPaper;
    MoveL Offs(pOrigin,281.88,309.94,0.00),v40,fine,tPen\WObj:=wPaper;
    MoveL Offs(pOrigin,281.88,309.94,6.00),v60,z5,tPen\WObj:=wPaper;
    MoveL Offs(pOrigin,283.36,308.24,6.00),vTravel,z5,tPen\WObj:=wPaper;
    MoveL Offs(pOrigin,283.36,308.24,0.00),v60,z0,tPen\WObj:=wPaper;
    MoveL Offs(pOrigin,281.02,308.45,0.00),v40,z0,tPen\WObj:=wPaper;
    MoveL Offs(pOrigin,279.11,308.24,0.00),v40,z0,tPen\WObj:=wPaper;
    MoveL Offs(pOrigin,278.48,307.81,0.00),v40,z0,tPen\WObj:=wPaper;
    MoveL Offs(pOrigin,278.48,307.81,0.00),v40,z0,tPen\WObj:=wPaper;
    MoveL Offs(pOrigin,278.48,308.02,0.00),v40,z0,tPen\WObj:=wPaper;
    MoveL Offs(pOrigin,277.41,307.81,0.00),v40,z0,tPen\WObj:=wPaper;
    MoveL Offs(pOrigin,277.20,308.24,0.00),v40,fine,tPen\WObj:=wPaper;
    MoveL Offs(pOrigin,277.20,308.24,6.00),v60,z5,tPen\WObj:=wPaper;
    MoveL Offs(pOrigin,278.48,307.81,6.00),vTravel,z5,tPen\WObj:=wPaper;
    MoveL Offs(pOrigin,278.48,307.81,0.00),v60,z0,tPen\WObj:=wPaper;
    MoveL Offs(pOrigin,278.90,307.25,0.00),v40,z0,tPen\WObj:=wPaper;
    MoveL Offs(pOrigin,282.73,306.18,0.00),v40,z0,tPen\WObj:=wPaper;
    MoveL Offs(pOrigin,284.21,305.26,0.00),v40,z0,tPen\WObj:=wPaper;
    MoveL Offs(pOrigin,283.36,305.90,0.00),v40,z0,tPen\WObj:=wPaper;
    MoveL Offs(pOrigin,283.79,305.69,0.00),v40,z0,tPen\WObj:=wPaper;
    MoveL Offs(pOrigin,283.36,305.90,0.00),v40,fine,tPen\WObj:=wPaper;
    MoveL Offs(pOrigin,283.36,305.90,6.00),v60,z5,tPen\WObj:=wPaper;
    MoveL Offs(pOrigin,286.55,306.75,6.00),vTravel,z5,tPen\WObj:=wPaper;
    MoveL Offs(pOrigin,286.55,306.75,0.00),v60,z0,tPen\WObj:=wPaper;
    MoveL Offs(pOrigin,287.19,305.69,0.00),v40,z0,tPen\WObj:=wPaper;
    MoveL Offs(pOrigin,287.83,305.69,0.00),v40,z0,tPen\WObj:=wPaper;
    MoveL Offs(pOrigin,287.83,305.69,0.00),v40,z0,tPen\WObj:=wPaper;
    MoveL Offs(pOrigin,287.83,306.75,0.00),v40,z0,tPen\WObj:=wPaper;
    MoveL Offs(pOrigin,287.12,308.80,0.00),v40,z0,tPen\WObj:=wPaper;
    MoveL Offs(pOrigin,285.70,309.94,0.00),v40,fine,tPen\WObj:=wPaper;
    MoveL Offs(pOrigin,285.70,309.94,6.00),v60,z5,tPen\WObj:=wPaper;
    MoveL Offs(pOrigin,286.55,311.21,6.00),vTravel,z5,tPen\WObj:=wPaper;
    MoveL Offs(pOrigin,286.55,311.21,0.00),v60,z0,tPen\WObj:=wPaper;
    MoveL Offs(pOrigin,284.42,312.27,0.00),v40,z0,tPen\WObj:=wPaper;
    MoveL Offs(pOrigin,282.73,312.27,0.00),v40,z0,tPen\WObj:=wPaper;
    MoveL Offs(pOrigin,277.41,310.79,0.00),v40,z0,tPen\WObj:=wPaper;
    MoveL Offs(pOrigin,275.92,311.00,0.00),v40,z0,tPen\WObj:=wPaper;
    MoveL Offs(pOrigin,275.92,311.00,0.00),v40,z0,tPen\WObj:=wPaper;
    MoveL Offs(pOrigin,276.56,311.64,0.00),v40,fine,tPen\WObj:=wPaper;
    MoveL Offs(pOrigin,276.56,311.64,6.00),v60,z5,tPen\WObj:=wPaper;
    MoveL Offs(pOrigin,274.01,307.17,6.00),vTravel,z5,tPen\WObj:=wPaper;
    MoveL Offs(pOrigin,274.01,307.17,0.00),v60,z0,tPen\WObj:=wPaper;
    MoveL Offs(pOrigin,272.10,306.96,0.00),v40,z0,tPen\WObj:=wPaper;
    MoveL Offs(pOrigin,269.55,307.60,0.00),v40,z0,tPen\WObj:=wPaper;
    MoveL Offs(pOrigin,267.42,307.60,0.00),v40,fine,tPen\WObj:=wPaper;
    MoveL Offs(pOrigin,267.42,307.60,6.00),v60,z5,tPen\WObj:=wPaper;
    MoveL Offs(pOrigin,274.01,307.17,6.00),vTravel,z5,tPen\WObj:=wPaper;
    MoveL Offs(pOrigin,274.01,307.17,0.00),v60,z0,tPen\WObj:=wPaper;
    MoveL Offs(pOrigin,274.65,306.18,0.00),v40,z0,tPen\WObj:=wPaper;
    MoveL Offs(pOrigin,276.77,305.48,0.00),v40,z0,tPen\WObj:=wPaper;
    MoveL Offs(pOrigin,276.77,305.48,0.00),v40,z0,tPen\WObj:=wPaper;
    MoveL Offs(pOrigin,278.48,305.48,0.00),v40,z0,tPen\WObj:=wPaper;
    MoveL Offs(pOrigin,278.48,305.48,0.00),v40,z0,tPen\WObj:=wPaper;
    MoveL Offs(pOrigin,279.54,305.48,0.00),v40,z0,tPen\WObj:=wPaper;
    MoveL Offs(pOrigin,282.73,304.27,0.00),v40,z0,tPen\WObj:=wPaper;
    MoveL Offs(pOrigin,285.06,302.50,0.00),v40,z0,tPen\WObj:=wPaper;
    MoveL Offs(pOrigin,285.49,302.29,0.00),v40,z0,tPen\WObj:=wPaper;
    MoveL Offs(pOrigin,287.40,300.16,0.00),v40,z0,tPen\WObj:=wPaper;
    MoveL Offs(pOrigin,288.67,299.38,0.00),v40,z0,tPen\WObj:=wPaper;
    MoveL Offs(pOrigin,291.23,299.10,0.00),v40,z0,tPen\WObj:=wPaper;
    MoveL Offs(pOrigin,291.86,299.74,0.00),v40,z0,tPen\WObj:=wPaper;
    MoveL Offs(pOrigin,291.86,299.74,0.00),v40,z0,tPen\WObj:=wPaper;
    MoveL Offs(pOrigin,293.14,299.74,0.00),v40,z0,tPen\WObj:=wPaper;
    MoveL Offs(pOrigin,293.77,300.38,0.00),v40,z0,tPen\WObj:=wPaper;
    MoveL Offs(pOrigin,293.35,299.74,0.00),v40,z0,tPen\WObj:=wPaper;
    MoveL Offs(pOrigin,294.41,300.66,0.00),v40,z0,tPen\WObj:=wPaper;
    MoveL Offs(pOrigin,296.11,300.80,0.00),v40,z0,tPen\WObj:=wPaper;
    MoveL Offs(pOrigin,296.11,299.74,0.00),v40,z0,tPen\WObj:=wPaper;
    MoveL Offs(pOrigin,293.77,299.10,0.00),v40,z0,tPen\WObj:=wPaper;
    MoveL Offs(pOrigin,293.77,299.10,0.00),v40,z0,tPen\WObj:=wPaper;
    MoveL Offs(pOrigin,292.92,297.83,0.00),v40,z0,tPen\WObj:=wPaper;
    MoveL Offs(pOrigin,292.29,297.83,0.00),v40,fine,tPen\WObj:=wPaper;
    MoveL Offs(pOrigin,292.29,297.83,6.00),v60,z5,tPen\WObj:=wPaper;
    MoveL Offs(pOrigin,292.50,295.91,6.00),vTravel,z5,tPen\WObj:=wPaper;
    MoveL Offs(pOrigin,292.50,295.91,0.00),v60,z0,tPen\WObj:=wPaper;
    MoveL Offs(pOrigin,289.31,297.33,0.00),v40,z0,tPen\WObj:=wPaper;
    MoveL Offs(pOrigin,286.34,299.74,0.00),v40,z0,tPen\WObj:=wPaper;
    MoveL Offs(pOrigin,285.91,299.95,0.00),v40,z0,tPen\WObj:=wPaper;
    MoveL Offs(pOrigin,278.90,304.62,0.00),v40,z0,tPen\WObj:=wPaper;
    MoveL Offs(pOrigin,278.48,305.48,0.00),v40,fine,tPen\WObj:=wPaper;
    MoveL Offs(pOrigin,278.48,305.48,6.00),v60,z5,tPen\WObj:=wPaper;
    MoveL Offs(pOrigin,279.54,302.29,6.00),vTravel,z5,tPen\WObj:=wPaper;
    MoveL Offs(pOrigin,279.54,302.29,0.00),v60,z0,tPen\WObj:=wPaper;
    MoveL Offs(pOrigin,279.33,302.50,0.00),v40,z0,tPen\WObj:=wPaper;
    MoveL Offs(pOrigin,280.39,301.65,0.00),v40,z0,tPen\WObj:=wPaper;
    MoveL Offs(pOrigin,280.39,301.65,0.00),v40,z0,tPen\WObj:=wPaper;
    MoveL Offs(pOrigin,281.66,301.23,0.00),v40,z0,tPen\WObj:=wPaper;
    MoveL Offs(pOrigin,283.79,299.31,0.00),v40,z0,tPen\WObj:=wPaper;
    MoveL Offs(pOrigin,285.49,296.98,0.00),v40,z0,tPen\WObj:=wPaper;
    MoveL Offs(pOrigin,287.61,295.49,0.00),v40,fine,tPen\WObj:=wPaper;
    MoveL Offs(pOrigin,287.61,295.49,6.00),v60,z5,tPen\WObj:=wPaper;
    MoveL Offs(pOrigin,287.61,294.21,6.00),vTravel,z5,tPen\WObj:=wPaper;
    MoveL Offs(pOrigin,287.61,294.21,0.00),v60,z0,tPen\WObj:=wPaper;
    MoveL Offs(pOrigin,286.55,294.28,0.00),v40,z0,tPen\WObj:=wPaper;
    MoveL Offs(pOrigin,282.09,298.25,0.00),v40,z0,tPen\WObj:=wPaper;
    MoveL Offs(pOrigin,279.75,299.74,0.00),v40,fine,tPen\WObj:=wPaper;
    MoveL Offs(pOrigin,279.75,299.74,6.00),v60,z5,tPen\WObj:=wPaper;
    MoveL Offs(pOrigin,281.66,299.52,6.00),vTravel,z5,tPen\WObj:=wPaper;
    MoveL Offs(pOrigin,281.66,299.52,0.00),v60,z0,tPen\WObj:=wPaper;
    MoveL Offs(pOrigin,280.60,300.80,0.00),v40,z0,tPen\WObj:=wPaper;
    MoveL Offs(pOrigin,280.39,301.65,0.00),v40,fine,tPen\WObj:=wPaper;
    MoveL Offs(pOrigin,280.39,301.65,6.00),v60,z5,tPen\WObj:=wPaper;
  ENDPROC

  PROC DrawPart33()
    MoveL Offs(pOrigin,286.34,301.23,6.00),vTravel,z5,tPen\WObj:=wPaper;
    MoveL Offs(pOrigin,286.34,301.23,0.00),v60,z0,tPen\WObj:=wPaper;
    MoveL Offs(pOrigin,286.12,301.65,0.00),v40,z0,tPen\WObj:=wPaper;
    MoveL Offs(pOrigin,286.34,301.23,0.00),v40,fine,tPen\WObj:=wPaper;
    MoveL Offs(pOrigin,286.34,301.23,6.00),v60,z5,tPen\WObj:=wPaper;
    MoveL Offs(pOrigin,287.19,303.14,6.00),vTravel,z5,tPen\WObj:=wPaper;
    MoveL Offs(pOrigin,287.19,303.14,0.00),v60,z0,tPen\WObj:=wPaper;
    MoveL Offs(pOrigin,286.98,303.56,0.00),v40,z0,tPen\WObj:=wPaper;
    MoveL Offs(pOrigin,287.19,303.14,0.00),v40,z0,tPen\WObj:=wPaper;
    MoveL Offs(pOrigin,286.98,303.56,0.00),v40,z0,tPen\WObj:=wPaper;
    MoveL Offs(pOrigin,287.61,302.71,0.00),v40,z0,tPen\WObj:=wPaper;
    MoveL Offs(pOrigin,288.89,302.50,0.00),v40,z0,tPen\WObj:=wPaper;
    MoveL Offs(pOrigin,288.89,302.50,0.00),v40,z0,tPen\WObj:=wPaper;
    MoveL Offs(pOrigin,289.95,301.01,0.00),v40,z0,tPen\WObj:=wPaper;
    MoveL Offs(pOrigin,290.38,300.80,0.00),v40,z0,tPen\WObj:=wPaper;
    MoveL Offs(pOrigin,290.16,301.01,0.00),v40,z0,tPen\WObj:=wPaper;
    MoveL Offs(pOrigin,290.38,300.59,0.00),v40,z0,tPen\WObj:=wPaper;
    MoveL Offs(pOrigin,291.86,299.74,0.00),v40,fine,tPen\WObj:=wPaper;
    MoveL Offs(pOrigin,291.86,299.74,6.00),v60,z5,tPen\WObj:=wPaper;
    MoveL Offs(pOrigin,290.80,300.59,6.00),vTravel,z5,tPen\WObj:=wPaper;
    MoveL Offs(pOrigin,290.80,300.59,0.00),v60,z0,tPen\WObj:=wPaper;
    MoveL Offs(pOrigin,291.23,300.38,0.00),v40,z0,tPen\WObj:=wPaper;
    MoveL Offs(pOrigin,290.80,300.59,0.00),v40,fine,tPen\WObj:=wPaper;
    MoveL Offs(pOrigin,290.80,300.59,6.00),v60,z5,tPen\WObj:=wPaper;
    MoveL Offs(pOrigin,290.80,302.50,6.00),vTravel,z5,tPen\WObj:=wPaper;
    MoveL Offs(pOrigin,290.80,302.50,0.00),v60,z0,tPen\WObj:=wPaper;
    MoveL Offs(pOrigin,291.44,302.08,0.00),v40,z0,tPen\WObj:=wPaper;
    MoveL Offs(pOrigin,293.14,301.86,0.00),v40,z0,tPen\WObj:=wPaper;
    MoveL Offs(pOrigin,294.41,303.07,0.00),v40,z0,tPen\WObj:=wPaper;
    MoveL Offs(pOrigin,295.69,303.14,0.00),v40,fine,tPen\WObj:=wPaper;
    MoveL Offs(pOrigin,295.69,303.14,6.00),v60,z5,tPen\WObj:=wPaper;
    MoveL Offs(pOrigin,294.20,303.14,6.00),vTravel,z5,tPen\WObj:=wPaper;
    MoveL Offs(pOrigin,294.20,303.14,0.00),v60,z0,tPen\WObj:=wPaper;
    MoveL Offs(pOrigin,293.07,304.62,0.00),v40,z0,tPen\WObj:=wPaper;
    MoveL Offs(pOrigin,293.56,306.33,0.00),v40,fine,tPen\WObj:=wPaper;
    MoveL Offs(pOrigin,293.56,306.33,6.00),v60,z5,tPen\WObj:=wPaper;
    MoveL Offs(pOrigin,292.92,304.84,6.00),vTravel,z5,tPen\WObj:=wPaper;
    MoveL Offs(pOrigin,292.92,304.84,0.00),v60,z0,tPen\WObj:=wPaper;
    MoveL Offs(pOrigin,291.44,305.33,0.00),v40,z0,tPen\WObj:=wPaper;
    MoveL Offs(pOrigin,291.01,306.54,0.00),v40,fine,tPen\WObj:=wPaper;
    MoveL Offs(pOrigin,291.01,306.54,6.00),v60,z5,tPen\WObj:=wPaper;
    MoveL Offs(pOrigin,287.83,305.69,6.00),vTravel,z5,tPen\WObj:=wPaper;
    MoveL Offs(pOrigin,287.83,305.69,0.00),v60,z0,tPen\WObj:=wPaper;
    MoveL Offs(pOrigin,288.89,303.14,0.00),v40,z0,tPen\WObj:=wPaper;
    MoveL Offs(pOrigin,288.89,303.14,0.00),v40,z0,tPen\WObj:=wPaper;
    MoveL Offs(pOrigin,289.74,303.14,0.00),v40,z0,tPen\WObj:=wPaper;
    MoveL Offs(pOrigin,290.38,302.71,0.00),v40,fine,tPen\WObj:=wPaper;
    MoveL Offs(pOrigin,290.38,302.71,6.00),v60,z5,tPen\WObj:=wPaper;
    MoveL Offs(pOrigin,287.19,299.10,6.00),vTravel,z5,tPen\WObj:=wPaper;
    MoveL Offs(pOrigin,287.19,299.10,0.00),v60,z0,tPen\WObj:=wPaper;
    MoveL Offs(pOrigin,287.61,298.67,0.00),v40,z0,tPen\WObj:=wPaper;
    MoveL Offs(pOrigin,287.19,299.10,0.00),v40,fine,tPen\WObj:=wPaper;
    MoveL Offs(pOrigin,287.19,299.10,6.00),v60,z5,tPen\WObj:=wPaper;
    MoveL Offs(pOrigin,287.61,294.21,6.00),vTravel,z5,tPen\WObj:=wPaper;
    MoveL Offs(pOrigin,287.61,294.21,0.00),v60,z0,tPen\WObj:=wPaper;
    MoveL Offs(pOrigin,290.16,293.15,0.00),v40,z0,tPen\WObj:=wPaper;
    MoveL Offs(pOrigin,294.41,293.36,0.00),v40,z0,tPen\WObj:=wPaper;
    MoveL Offs(pOrigin,294.41,293.36,0.00),v40,z0,tPen\WObj:=wPaper;
    MoveL Offs(pOrigin,294.20,291.45,0.00),v40,z0,tPen\WObj:=wPaper;
    MoveL Offs(pOrigin,294.20,291.45,0.00),v40,z0,tPen\WObj:=wPaper;
    MoveL Offs(pOrigin,294.62,291.24,0.00),v40,z0,tPen\WObj:=wPaper;
    MoveL Offs(pOrigin,296.89,291.88,0.00),v40,z0,tPen\WObj:=wPaper;
    MoveL Offs(pOrigin,296.75,293.36,0.00),v40,z0,tPen\WObj:=wPaper;
    MoveL Offs(pOrigin,296.33,294.00,0.00),v40,z0,tPen\WObj:=wPaper;
    MoveL Offs(pOrigin,296.33,294.00,0.00),v40,z0,tPen\WObj:=wPaper;
    MoveL Offs(pOrigin,296.75,295.27,0.00),v40,z0,tPen\WObj:=wPaper;
    MoveL Offs(pOrigin,296.54,297.40,0.00),v40,fine,tPen\WObj:=wPaper;
    MoveL Offs(pOrigin,296.54,297.40,6.00),v60,z5,tPen\WObj:=wPaper;
    MoveL Offs(pOrigin,296.33,294.00,6.00),vTravel,z5,tPen\WObj:=wPaper;
    MoveL Offs(pOrigin,296.33,294.00,0.00),v60,z0,tPen\WObj:=wPaper;
    MoveL Offs(pOrigin,294.41,293.36,0.00),v40,fine,tPen\WObj:=wPaper;
    MoveL Offs(pOrigin,294.41,293.36,6.00),v60,z5,tPen\WObj:=wPaper;
    MoveL Offs(pOrigin,294.20,291.45,6.00),vTravel,z5,tPen\WObj:=wPaper;
    MoveL Offs(pOrigin,294.20,291.45,0.00),v60,z0,tPen\WObj:=wPaper;
    MoveL Offs(pOrigin,292.50,290.60,0.00),v40,z0,tPen\WObj:=wPaper;
    MoveL Offs(pOrigin,290.38,290.39,0.00),v40,z0,tPen\WObj:=wPaper;
    MoveL Offs(pOrigin,289.52,289.96,0.00),v40,z0,tPen\WObj:=wPaper;
    MoveL Offs(pOrigin,287.40,290.39,0.00),v40,z0,tPen\WObj:=wPaper;
    MoveL Offs(pOrigin,286.62,289.96,0.00),v40,z0,tPen\WObj:=wPaper;
    MoveL Offs(pOrigin,287.19,289.11,0.00),v40,z0,tPen\WObj:=wPaper;
    MoveL Offs(pOrigin,288.46,288.40,0.00),v40,z0,tPen\WObj:=wPaper;
    MoveL Offs(pOrigin,292.92,287.62,0.00),v40,z0,tPen\WObj:=wPaper;
    MoveL Offs(pOrigin,292.92,287.62,0.00),v40,z0,tPen\WObj:=wPaper;
    MoveL Offs(pOrigin,295.90,288.90,0.00),v40,z0,tPen\WObj:=wPaper;
    MoveL Offs(pOrigin,296.75,289.11,0.00),v40,z0,tPen\WObj:=wPaper;
    MoveL Offs(pOrigin,296.96,291.66,0.00),v40,fine,tPen\WObj:=wPaper;
    MoveL Offs(pOrigin,296.96,291.66,6.00),v60,z5,tPen\WObj:=wPaper;
    MoveL Offs(pOrigin,296.75,289.11,6.00),vTravel,z5,tPen\WObj:=wPaper;
    MoveL Offs(pOrigin,296.75,289.11,0.00),v60,z0,tPen\WObj:=wPaper;
    MoveL Offs(pOrigin,297.60,288.26,0.00),v40,z0,tPen\WObj:=wPaper;
    MoveL Offs(pOrigin,297.17,284.23,0.00),v40,z0,tPen\WObj:=wPaper;
    MoveL Offs(pOrigin,297.17,284.23,0.00),v40,z0,tPen\WObj:=wPaper;
    MoveL Offs(pOrigin,297.10,283.16,0.00),v40,z0,tPen\WObj:=wPaper;
    MoveL Offs(pOrigin,295.90,281.67,0.00),v40,z0,tPen\WObj:=wPaper;
    MoveL Offs(pOrigin,295.90,281.67,0.00),v40,z0,tPen\WObj:=wPaper;
    MoveL Offs(pOrigin,292.92,279.90,0.00),v40,z0,tPen\WObj:=wPaper;
    MoveL Offs(pOrigin,290.80,279.34,0.00),v40,z0,tPen\WObj:=wPaper;
    MoveL Offs(pOrigin,287.83,279.76,0.00),v40,z0,tPen\WObj:=wPaper;
    MoveL Offs(pOrigin,287.19,280.61,0.00),v40,z0,tPen\WObj:=wPaper;
    MoveL Offs(pOrigin,287.19,280.61,0.00),v40,z0,tPen\WObj:=wPaper;
    MoveL Offs(pOrigin,287.83,281.04,0.00),v40,z0,tPen\WObj:=wPaper;
    MoveL Offs(pOrigin,290.16,281.04,0.00),v40,z0,tPen\WObj:=wPaper;
    MoveL Offs(pOrigin,290.80,281.60,0.00),v40,z0,tPen\WObj:=wPaper;
    MoveL Offs(pOrigin,292.71,282.03,0.00),v40,z0,tPen\WObj:=wPaper;
    MoveL Offs(pOrigin,297.17,284.23,0.00),v40,fine,tPen\WObj:=wPaper;
    MoveL Offs(pOrigin,297.17,284.23,6.00),v60,z5,tPen\WObj:=wPaper;
    MoveL Offs(pOrigin,297.17,282.95,6.00),vTravel,z5,tPen\WObj:=wPaper;
    MoveL Offs(pOrigin,297.17,282.95,0.00),v60,z0,tPen\WObj:=wPaper;
    MoveL Offs(pOrigin,296.54,282.31,0.00),v40,z0,tPen\WObj:=wPaper;
    MoveL Offs(pOrigin,296.54,281.46,0.00),v40,z0,tPen\WObj:=wPaper;
    MoveL Offs(pOrigin,297.39,282.10,0.00),v40,z0,tPen\WObj:=wPaper;
    MoveL Offs(pOrigin,298.24,281.67,0.00),v40,z0,tPen\WObj:=wPaper;
    MoveL Offs(pOrigin,298.66,281.89,0.00),v40,z0,tPen\WObj:=wPaper;
    MoveL Offs(pOrigin,298.66,282.74,0.00),v40,fine,tPen\WObj:=wPaper;
    MoveL Offs(pOrigin,298.66,282.74,6.00),v60,z5,tPen\WObj:=wPaper;
    MoveL Offs(pOrigin,296.75,289.11,6.00),vTravel,z5,tPen\WObj:=wPaper;
    MoveL Offs(pOrigin,296.75,289.11,0.00),v60,z0,tPen\WObj:=wPaper;
    MoveL Offs(pOrigin,295.97,288.69,0.00),v40,z0,tPen\WObj:=wPaper;
    MoveL Offs(pOrigin,295.76,287.20,0.00),v40,z0,tPen\WObj:=wPaper;
    MoveL Offs(pOrigin,295.05,286.14,0.00),v40,z0,tPen\WObj:=wPaper;
  ENDPROC

  PROC DrawPart34()
    MoveL Offs(pOrigin,293.77,285.15,0.00),v40,z0,tPen\WObj:=wPaper;
    MoveL Offs(pOrigin,292.50,284.65,0.00),v40,z0,tPen\WObj:=wPaper;
    MoveL Offs(pOrigin,289.31,284.44,0.00),v40,z0,tPen\WObj:=wPaper;
    MoveL Offs(pOrigin,287.40,285.15,0.00),v40,z0,tPen\WObj:=wPaper;
    MoveL Offs(pOrigin,286.98,285.92,0.00),v40,z0,tPen\WObj:=wPaper;
    MoveL Offs(pOrigin,286.98,285.92,0.00),v40,z0,tPen\WObj:=wPaper;
    MoveL Offs(pOrigin,287.61,286.35,0.00),v40,z0,tPen\WObj:=wPaper;
    MoveL Offs(pOrigin,290.59,286.14,0.00),v40,z0,tPen\WObj:=wPaper;
    MoveL Offs(pOrigin,291.86,286.35,0.00),v40,z0,tPen\WObj:=wPaper;
    MoveL Offs(pOrigin,292.92,287.62,0.00),v40,fine,tPen\WObj:=wPaper;
    MoveL Offs(pOrigin,292.92,287.62,6.00),v60,z5,tPen\WObj:=wPaper;
    MoveL Offs(pOrigin,287.19,286.35,6.00),vTravel,z5,tPen\WObj:=wPaper;
    MoveL Offs(pOrigin,287.19,286.35,0.00),v60,z0,tPen\WObj:=wPaper;
    MoveL Offs(pOrigin,286.55,286.07,0.00),v40,z0,tPen\WObj:=wPaper;
    MoveL Offs(pOrigin,284.21,287.48,0.00),v40,z0,tPen\WObj:=wPaper;
    MoveL Offs(pOrigin,283.79,288.62,0.00),v40,z0,tPen\WObj:=wPaper;
    MoveL Offs(pOrigin,282.51,289.11,0.00),v40,z0,tPen\WObj:=wPaper;
    MoveL Offs(pOrigin,282.94,288.90,0.00),v40,z0,tPen\WObj:=wPaper;
    MoveL Offs(pOrigin,282.94,287.84,0.00),v40,z0,tPen\WObj:=wPaper;
    MoveL Offs(pOrigin,284.00,287.41,0.00),v40,z0,tPen\WObj:=wPaper;
    MoveL Offs(pOrigin,283.15,287.84,0.00),v40,z0,tPen\WObj:=wPaper;
    MoveL Offs(pOrigin,283.58,287.62,0.00),v40,z0,tPen\WObj:=wPaper;
    MoveL Offs(pOrigin,283.15,287.84,0.00),v40,fine,tPen\WObj:=wPaper;
    MoveL Offs(pOrigin,283.15,287.84,6.00),v60,z5,tPen\WObj:=wPaper;
    MoveL Offs(pOrigin,281.24,288.48,6.00),vTravel,z5,tPen\WObj:=wPaper;
    MoveL Offs(pOrigin,281.24,288.48,0.00),v60,z0,tPen\WObj:=wPaper;
    MoveL Offs(pOrigin,279.54,290.60,0.00),v40,fine,tPen\WObj:=wPaper;
    MoveL Offs(pOrigin,279.54,290.60,6.00),v60,z5,tPen\WObj:=wPaper;
    MoveL Offs(pOrigin,279.54,292.09,6.00),vTravel,z5,tPen\WObj:=wPaper;
    MoveL Offs(pOrigin,279.54,292.09,0.00),v60,z0,tPen\WObj:=wPaper;
    MoveL Offs(pOrigin,279.33,292.51,0.00),v40,z0,tPen\WObj:=wPaper;
    MoveL Offs(pOrigin,279.54,292.09,0.00),v40,fine,tPen\WObj:=wPaper;
    MoveL Offs(pOrigin,279.54,292.09,6.00),v60,z5,tPen\WObj:=wPaper;
    MoveL Offs(pOrigin,278.69,293.36,6.00),vTravel,z5,tPen\WObj:=wPaper;
    MoveL Offs(pOrigin,278.69,293.36,0.00),v60,z0,tPen\WObj:=wPaper;
    MoveL Offs(pOrigin,280.39,291.02,0.00),v40,z0,tPen\WObj:=wPaper;
    MoveL Offs(pOrigin,281.24,290.39,0.00),v40,fine,tPen\WObj:=wPaper;
    MoveL Offs(pOrigin,281.24,290.39,6.00),v60,z5,tPen\WObj:=wPaper;
    MoveL Offs(pOrigin,281.24,291.88,6.00),vTravel,z5,tPen\WObj:=wPaper;
    MoveL Offs(pOrigin,281.24,291.88,0.00),v60,z0,tPen\WObj:=wPaper;
    MoveL Offs(pOrigin,281.02,292.30,0.00),v40,z0,tPen\WObj:=wPaper;
    MoveL Offs(pOrigin,281.24,291.88,0.00),v40,fine,tPen\WObj:=wPaper;
    MoveL Offs(pOrigin,281.24,291.88,6.00),v60,z5,tPen\WObj:=wPaper;
    MoveL Offs(pOrigin,278.69,289.11,6.00),vTravel,z5,tPen\WObj:=wPaper;
    MoveL Offs(pOrigin,278.69,289.11,0.00),v60,z0,tPen\WObj:=wPaper;
    MoveL Offs(pOrigin,281.24,285.71,0.00),v40,z0,tPen\WObj:=wPaper;
    MoveL Offs(pOrigin,282.73,285.08,0.00),v40,z0,tPen\WObj:=wPaper;
    MoveL Offs(pOrigin,282.94,285.08,0.00),v40,z0,tPen\WObj:=wPaper;
    MoveL Offs(pOrigin,283.79,285.08,0.00),v40,z0,tPen\WObj:=wPaper;
    MoveL Offs(pOrigin,285.27,284.01,0.00),v40,z0,tPen\WObj:=wPaper;
    MoveL Offs(pOrigin,285.70,283.80,0.00),v40,z0,tPen\WObj:=wPaper;
    MoveL Offs(pOrigin,287.19,282.88,0.00),v40,z0,tPen\WObj:=wPaper;
    MoveL Offs(pOrigin,290.59,281.67,0.00),v40,fine,tPen\WObj:=wPaper;
    MoveL Offs(pOrigin,290.59,281.67,6.00),v60,z5,tPen\WObj:=wPaper;
    MoveL Offs(pOrigin,287.40,281.04,6.00),vTravel,z5,tPen\WObj:=wPaper;
    MoveL Offs(pOrigin,287.40,281.04,0.00),v60,z0,tPen\WObj:=wPaper;
    MoveL Offs(pOrigin,286.98,280.61,0.00),v40,z0,tPen\WObj:=wPaper;
    MoveL Offs(pOrigin,286.34,280.61,0.00),v40,fine,tPen\WObj:=wPaper;
    MoveL Offs(pOrigin,286.34,280.61,6.00),v60,z5,tPen\WObj:=wPaper;
    MoveL Offs(pOrigin,287.83,277.85,6.00),vTravel,z5,tPen\WObj:=wPaper;
    MoveL Offs(pOrigin,287.83,277.85,0.00),v60,z0,tPen\WObj:=wPaper;
    MoveL Offs(pOrigin,288.25,277.64,0.00),v40,z0,tPen\WObj:=wPaper;
    MoveL Offs(pOrigin,287.83,277.85,0.00),v40,fine,tPen\WObj:=wPaper;
    MoveL Offs(pOrigin,287.83,277.85,6.00),v60,z5,tPen\WObj:=wPaper;
    MoveL Offs(pOrigin,285.49,276.58,6.00),vTravel,z5,tPen\WObj:=wPaper;
    MoveL Offs(pOrigin,285.49,276.58,0.00),v60,z0,tPen\WObj:=wPaper;
    MoveL Offs(pOrigin,285.06,276.58,0.00),v40,z0,tPen\WObj:=wPaper;
    MoveL Offs(pOrigin,284.85,277.00,0.00),v40,z0,tPen\WObj:=wPaper;
    MoveL Offs(pOrigin,284.85,277.42,0.00),v40,z0,tPen\WObj:=wPaper;
    MoveL Offs(pOrigin,284.21,277.07,0.00),v40,z0,tPen\WObj:=wPaper;
    MoveL Offs(pOrigin,282.30,277.64,0.00),v40,fine,tPen\WObj:=wPaper;
    MoveL Offs(pOrigin,282.30,277.64,6.00),v60,z5,tPen\WObj:=wPaper;
    MoveL Offs(pOrigin,281.45,278.49,6.00),vTravel,z5,tPen\WObj:=wPaper;
    MoveL Offs(pOrigin,281.45,278.49,0.00),v60,z0,tPen\WObj:=wPaper;
    MoveL Offs(pOrigin,280.60,278.49,0.00),v40,z0,tPen\WObj:=wPaper;
    MoveL Offs(pOrigin,279.96,279.34,0.00),v40,fine,tPen\WObj:=wPaper;
    MoveL Offs(pOrigin,279.96,279.34,6.00),v60,z5,tPen\WObj:=wPaper;
    MoveL Offs(pOrigin,281.45,279.76,6.00),vTravel,z5,tPen\WObj:=wPaper;
    MoveL Offs(pOrigin,281.45,279.76,0.00),v60,z0,tPen\WObj:=wPaper;
    MoveL Offs(pOrigin,280.53,280.19,0.00),v40,z0,tPen\WObj:=wPaper;
    MoveL Offs(pOrigin,279.11,282.74,0.00),v40,fine,tPen\WObj:=wPaper;
    MoveL Offs(pOrigin,279.11,282.74,6.00),v60,z5,tPen\WObj:=wPaper;
    MoveL Offs(pOrigin,279.33,273.17,6.00),vTravel,z5,tPen\WObj:=wPaper;
    MoveL Offs(pOrigin,279.33,273.17,0.00),v60,z0,tPen\WObj:=wPaper;
    MoveL Offs(pOrigin,279.25,271.90,0.00),v40,z0,tPen\WObj:=wPaper;
    MoveL Offs(pOrigin,277.41,271.05,0.00),v40,fine,tPen\WObj:=wPaper;
    MoveL Offs(pOrigin,277.41,271.05,6.00),v60,z5,tPen\WObj:=wPaper;
    MoveL Offs(pOrigin,276.35,269.35,6.00),vTravel,z5,tPen\WObj:=wPaper;
    MoveL Offs(pOrigin,276.35,269.35,0.00),v60,z0,tPen\WObj:=wPaper;
    MoveL Offs(pOrigin,277.20,270.06,0.00),v40,z0,tPen\WObj:=wPaper;
    MoveL Offs(pOrigin,279.54,270.84,0.00),v40,z0,tPen\WObj:=wPaper;
    MoveL Offs(pOrigin,279.33,271.69,0.00),v40,z0,tPen\WObj:=wPaper;
    MoveL Offs(pOrigin,279.54,271.05,0.00),v40,z0,tPen\WObj:=wPaper;
    MoveL Offs(pOrigin,279.96,270.84,0.00),v40,z0,tPen\WObj:=wPaper;
    MoveL Offs(pOrigin,283.36,271.05,0.00),v40,z0,tPen\WObj:=wPaper;
    MoveL Offs(pOrigin,284.85,270.62,0.00),v40,fine,tPen\WObj:=wPaper;
    MoveL Offs(pOrigin,284.85,270.62,6.00),v60,z5,tPen\WObj:=wPaper;
    MoveL Offs(pOrigin,284.42,272.11,6.00),vTravel,z5,tPen\WObj:=wPaper;
    MoveL Offs(pOrigin,284.42,272.11,0.00),v60,z0,tPen\WObj:=wPaper;
    MoveL Offs(pOrigin,280.81,271.90,0.00),v40,fine,tPen\WObj:=wPaper;
    MoveL Offs(pOrigin,280.81,271.90,6.00),v60,z5,tPen\WObj:=wPaper;
    MoveL Offs(pOrigin,279.33,273.17,6.00),vTravel,z5,tPen\WObj:=wPaper;
    MoveL Offs(pOrigin,279.33,273.17,0.00),v60,z0,tPen\WObj:=wPaper;
    MoveL Offs(pOrigin,282.30,273.17,0.00),v40,z0,tPen\WObj:=wPaper;
    MoveL Offs(pOrigin,283.15,274.02,0.00),v40,z0,tPen\WObj:=wPaper;
    MoveL Offs(pOrigin,283.15,274.02,0.00),v40,z0,tPen\WObj:=wPaper;
    MoveL Offs(pOrigin,282.51,273.39,0.00),v40,fine,tPen\WObj:=wPaper;
    MoveL Offs(pOrigin,282.51,273.39,6.00),v60,z5,tPen\WObj:=wPaper;
    MoveL Offs(pOrigin,279.33,273.17,6.00),vTravel,z5,tPen\WObj:=wPaper;
    MoveL Offs(pOrigin,279.33,273.17,0.00),v60,z0,tPen\WObj:=wPaper;
    MoveL Offs(pOrigin,275.08,272.75,0.00),v40,fine,tPen\WObj:=wPaper;
    MoveL Offs(pOrigin,275.08,272.75,6.00),v60,z5,tPen\WObj:=wPaper;
    MoveL Offs(pOrigin,270.83,271.69,6.00),vTravel,z5,tPen\WObj:=wPaper;
    MoveL Offs(pOrigin,270.83,271.69,0.00),v60,z0,tPen\WObj:=wPaper;
    MoveL Offs(pOrigin,268.27,273.17,0.00),v40,z0,tPen\WObj:=wPaper;
    MoveL Offs(pOrigin,263.60,273.39,0.00),v40,z0,tPen\WObj:=wPaper;
    MoveL Offs(pOrigin,249.57,270.70,0.00),v40,z0,tPen\WObj:=wPaper;
    MoveL Offs(pOrigin,247.88,269.77,0.00),v40,z0,tPen\WObj:=wPaper;
    MoveL Offs(pOrigin,246.74,268.29,0.00),v40,z0,tPen\WObj:=wPaper;
    MoveL Offs(pOrigin,246.60,265.74,0.00),v40,z0,tPen\WObj:=wPaper;
  ENDPROC

